Yaskawa INFORM job: OK_R2_O8A-O21A(90,0)OKKR.JBI

/JOB
//NAME OK_R2_O8A-O21A(90,0)OKKR
///FOLDERNAME X4
//POS
///NPOS 663,663,663,26,0,0
///TOOL 0
///POSTYPE PULSE
///PULSE
C00000=132511,-103668,-126871,-1472,79341,68717
C00001=132511,-105453,-125920,-1479,77839,68735
C00002=149942,-121925,-119361,5630,57848,69572
C00003=131289,-120708,-115141,16553,58451,62255
C00004=130492,-107448,-108919,16502,61476,62404
C00005=130492,-107531,-107691,16624,60708,62286
C00006=130492,-107522,-107880,16606,60824,62304
C00007=130122,-101219,-105586,16530,62651,62436
C00008=130467,-107013,-108826,16492,61638,62417
C00009=173804,-84257,-100337,-8034,65857,78258
C00010=173658,-84030,-99866,-7982,65672,78220
C00011=173658,-84451,-98929,-8028,64885,78273
C00012=173658,-84370,-99117,-8019,65041,78263
C00013=172100,-80256,-97322,-7106,65901,77657
C00014=174189,-84275,-102553,-8181,67232,78295
C00015=146680,-106555,-114552,7207,63010,68642
C00016=194694,-79170,-110255,25784,98520,-48468
C00017=198558,-80793,-107909,24687,95396,-47836
C00018=200090,-81195,-106872,24266,94212,-47563
C00019=202263,-84154,-108139,23691,92956,-47080
C00020=202263,-85492,-106716,23644,91519,-47366
C00021=203864,-86202,-108997,23266,92055,-46716
C00022=200090,-81195,-106872,24266,94212,-47563
C00023=174358,-91389,-89628,58384,85447,-80654
C00024=175228,-93280,-90391,58296,84646,-80691
C00025=174358,-91389,-89628,58384,85447,-80654
C00026=168427,-86826,-93699,59246,91643,-79819
C00027=162839,-83719,-106729,43881,81993,-66911
C00028=147123,-91237,-114479,20257,52031,-49855
C00029=112908,-124838,-130477,22240,82773,-36203
C00030=117493,-120147,-121828,21064,78888,-35282
C00031=131517,-88028,-114974,8271,96172,-30135
C00032=131517,-89283,-114090,8245,94996,-30214
C00033=131517,-88930,-114352,8253,95335,-30191
C00034=131178,-82908,-111873,8367,96921,-30191
C00035=131517,-87249,-115462,8285,96867,-30089
C00036=132831,-90163,-114266,11578,93705,-29175
C00037=134095,-89636,-114054,11263,93680,-28777
C00038=131312,-89742,-115220,11972,94693,-29560
C00039=110699,-95947,-121920,22827,92218,-35184
C00040=159423,-136044,-122705,19473,51748,-49954
C00041=156084,-144100,-135379,20578,56007,-50549
C00042=159635,-139405,-132559,18260,112136,-84879
C00043=178843,-153016,-133090,20490,101295,-79475
C00044=178843,-153131,-133279,20494,101347,-79466
C00045=178843,-151887,-131264,20445,100783,-79562
C00046=178843,-153131,-133279,20494,101347,-79466
C00047=178681,-162456,-135669,20227,98263,-80057
C00048=165549,-147119,-131679,18745,106518,-83551
C00049=164263,-165353,-136391,17937,100651,-41944
C00050=168242,-162829,-132237,18538,98565,-40818
C00051=170474,-158220,-131092,19006,99630,-39839
C00052=168242,-162829,-132237,18538,98565,-40818
C00053=163940,-146805,-133599,18623,108164,-40895
C00054=162398,-133850,-130940,19068,113277,-40626
C00055=162571,-113567,-127717,17378,114163,-86924
C00056=160654,-117481,-127396,16916,112431,-87902
C00057=160654,-117651,-127195,16888,112229,-87933
C00058=160654,-118532,-125995,16733,111086,-88103
C00059=160654,-118346,-126273,16766,111343,-88065
C00060=161650,-123459,-127890,16641,109583,-87959
C00061=158594,-113131,-127392,17075,114977,-88272
C00062=174543,-100010,-122844,18621,115499,-82286
C00063=174543,-100010,-122844,18621,115499,-82286
C00064=174543,-100010,-122844,18621,115499,-22315
C00065=138816,-129701,-130055,13678,112254,-36070
C00066=137500,-131474,-125884,13183,109137,-36932
C00067=137500,-131471,-125777,13177,109074,-36939
C00068=139149,-130411,-125460,13458,109147,-36324
C00069=137500,-131471,-125777,13177,109074,-36939
C00070=137500,-129047,-134180,13875,115320,-36192
C00071=137500,-130207,-132407,13667,113680,-36396
C00072=137899,-129904,-132317,13740,113712,-36243
C00073=137899,-129904,-132317,13740,113712,-68510
C00074=153549,-123160,-126704,15778,110958,-63049
C00075=153549,-123239,-126516,15760,110807,-63070
C00076=153549,-123761,-124983,15622,109641,-63231
C00077=153549,-123239,-126516,15760,110807,-63070
C00078=162223,-110280,-122283,17095,113025,-59536
C00079=162223,-111585,-120346,16843,111240,-59807
C00080=163386,-116637,-122034,16744,109515,-59637
C00081=162108,-110157,-121578,17034,112692,-59632
C00082=164629,-100924,-122013,18009,116976,-58006
C00083=164629,-100924,-122013,18009,116976,-86315
C00084=167353,-101147,-115616,17756,113668,-85844
C00085=165427,-104649,-116407,17406,112807,-86697
C00086=165427,-101226,-120322,18070,116786,-86050
C00087=165427,-100996,-120510,18111,117009,-86012
C00088=148525,-143011,-136643,-3983,84771,6637
C00089=128066,-147732,-136598,-30045,86114,11272
C00090=107762,-175532,-134890,-18909,55578,-3499
C00091=107762,-174389,-134000,-18900,55616,-3506
C00092=107762,-171707,-131824,-18892,55653,-3513
C00093=107762,-174389,-134000,-18900,55616,-3506
C00094=110240,-168768,-132692,-19371,58166,-2939
C00095=107762,-174389,-134000,-18900,55616,-3506
C00096=136558,-139033,-124155,-30771,85335,13620
C00097=136645,-139245,-122439,-30816,84359,13917
C00098=135016,-140023,-122655,-30663,83532,13499
C00099=136645,-139245,-122439,-30816,84359,13917
C00100=136645,-142239,-130726,-30739,87441,13088
C00101=136645,-142239,-130726,-30739,87441,13088
C00102=136231,-126717,-125654,-30746,91494,11840
C00103=98133,-136848,-119853,8087,80711,399
C00104=120576,-107226,-130969,-4806,98429,-26759
C00105=134040,-103912,-127141,-12417,95216,-42526
C00106=135128,-102736,-122709,-12628,93295,-41985
C00107=135270,-98410,-119352,-12667,93467,-41957
C00108=135270,-99211,-118697,-12651,92671,-41876
C00109=135270,-98984,-118890,-12655,92901,-41899
C00110=134962,-94751,-117294,-12605,94023,-42111
C00111=135502,-100967,-121058,-12716,93242,-41857
C00112=134459,-102900,-122675,-12466,93098,-42180
C00113=132900,-95838,-124142,-12211,97313,-43092
C00114=133104,-101231,-126476,-12555,90730,-41824
C00115=142488,-103018,-116603,18920,70477,33231
C00116=149408,-93922,-109008,15541,69095,35470
C00117=149408,-94512,-107956,15635,68178,35347
C00118=149408,-94372,-108222,15611,68405,35378
C00119=148690,-90146,-106536,15855,69631,35290
C00120=149408,-93897,-109054,15536,69135,35476
C00121=123067,-90692,-110186,27168,77789,27787
C00122=102416,-91941,-110630,34518,86135,22666
C00123=101917,-92285,-106963,34730,79171,22421
C00124=101917,-92861,-105821,34832,78340,22159
C00125=102166,-91294,-105409,34682,78702,22372
C00126=102552,-87773,-103968,34461,79319,22719
C00127=102166,-90677,-106542,34586,79544,22637
C00128=123117,-127863,-126220,28315,69551,25784
C00129=125315,-122167,-126738,14196,74486,31169
C00130=125647,-109964,-126758,-6698,85320,36650
C00131=127309,-126191,-121158,-24496,77378,41430
C00132=122509,-120998,-116871,-23174,76039,39921
C00133=117160,-104372,-112630,-18566,82677,37125
C00134=117160,-104907,-110988,-18612,81456,37312
C00135=117160,-104733,-111581,-18595,81887,37246
C00136=112842,-111563,-113988,-14481,77147,33000
C00137=113063,-106504,-112219,-14479,78650,32898
C00138=112842,-111563,-113988,-14481,77147,33000
C00139=122612,-110522,-114147,-22924,79491,39282
C00140=127138,-114707,-118233,-24171,81082,40600
C00141=112168,-135147,-125869,-19703,71474,13622
C00142=107112,-124941,-122811,-17686,73526,11445
C00143=98892,-86649,-110918,-2998,94873,-14107
C00144=112057,-63273,-99647,-16927,107898,6848
C00145=111820,-63961,-99109,-16821,107199,6872
C00146=111820,-65039,-98309,-16715,106195,7017
C00147=111820,-64914,-98405,-16727,106313,7000
C00148=110559,-64565,-98232,-16557,106153,6607
C00149=111820,-64402,-98791,-16776,106793,6930
C00150=102401,-90236,-113117,129,94163,-18304
C00151=122722,-94557,-112635,-4536,92169,-11873
C00152=122722,-95060,-112012,-4533,91529,-11850
C00153=122722,-94938,-112169,-4534,91688,-11856
C00154=124421,-94788,-112110,-4914,91823,-11321
C00155=122722,-94458,-112752,-4538,92292,-11877
C00156=121995,-82445,-116286,-4470,100580,-12401
C00157=106227,-105095,-124470,409,77251,-17488
C00158=147196,-120547,-129970,14917,75808,-13222
C00159=161004,-130220,-121828,20444,67155,-12825
C00160=163784,-117907,-115753,19016,68936,-11464
C00161=172766,-99094,-111810,8888,79207,-7928
C00162=172766,-99537,-110960,8908,78464,-7982
C00163=164799,-113448,-113379,18515,69495,-10996
C00164=160173,-111708,-112729,20272,71037,-12446
C00165=159937,-107532,-111273,20230,72269,-12319
C00166=160173,-111708,-112729,20272,71037,-12446
C00167=157530,-113449,-113320,21331,71196,-13397
C00168=157502,-114878,-111335,21583,69377,-13748
C00169=159463,-112600,-110567,20755,69532,-12980
C00170=157502,-114878,-111335,21583,69377,-13748
C00171=157530,-113449,-113320,21331,71196,-13397
C00172=164799,-113448,-113379,18515,69495,-10996
C00173=163784,-117907,-115753,19016,68936,-11464
C00174=161004,-130220,-121828,20444,67155,-12825
C00175=158635,-143974,-124952,47178,64629,48132
C00176=161510,-136095,-119169,46184,63472,49060
C00177=162608,-132555,-115350,46042,62530,49158
C00178=162346,-131008,-113540,46239,62439,48970
C00179=162608,-133192,-116899,45817,62973,49385
C00180=136560,-74570,-80638,73986,100743,31924
C00181=136560,-74368,-74379,73183,99581,30233
C00182=138115,-75223,-74700,73053,98436,30293
C00183=135508,-73752,-74143,73275,100358,30196
C00184=149616,-145660,-96573,81184,49972,24507
C00185=150329,-142641,-96001,80244,49710,25268
C00186=148962,-149729,-97186,82532,50127,23453
C00187=146770,-153464,-99018,82858,51507,22849
C00188=140616,-162996,-103531,83341,55379,21287
C00189=129649,-178931,-115518,81569,62637,20208
C00190=149811,-117254,-127694,14309,93218,9052
C00191=138773,-86779,-112433,16512,101214,6420
C00192=139010,-84837,-109587,16423,100448,6393
C00193=139010,-86284,-108173,16326,98898,6181
C00194=139046,-85929,-108499,16342,99259,6242
C00195=139851,-81484,-106752,16280,100273,6644
C00196=139210,-85073,-109125,16364,100022,6400
C00197=160229,-93267,-112119,12359,94277,12585
C00198=159749,-92653,-111811,12461,94470,12448
C00199=159749,-93339,-110977,12438,93625,12360
C00200=159895,-92298,-111808,12436,94626,12511
C00201=160151,-89339,-110624,12406,95366,12669
C00202=159895,-92298,-111808,12436,94626,12511
C00203=154010,-101242,-121994,13665,97135,10872
C00204=154083,-100267,-121778,13665,97483,10934
C00205=147006,-81102,-116195,13282,100818,-40144
C00206=151269,-63896,-105225,12354,102282,-38687
C00207=152138,-63686,-103764,12097,101397,-38514
C00208=152138,-64898,-103136,12048,100410,-38612
C00209=152138,-64707,-103240,12056,100569,-38597
C00210=153752,-65312,-103536,11647,100239,-38140
C00211=152274,-63472,-103683,12067,101440,-38470
C00212=162010,-107602,-126737,9369,91949,-36281
C00213=162010,-107602,-126737,9369,91949,-36281
C00214=210314,-79584,-107375,-35746,108623,54127
C00215=185587,-33049,-75742,-32288,103518,46434
C00216=184078,-34029,-75535,-31853,102480,46201
C00217=182552,-34930,-76118,-31484,101891,45830
C00218=182816,-34825,-76051,-31547,101988,45895
C00219=182831,-36048,-74896,-31379,100842,46225
C00220=185721,-33305,-75942,-32316,103553,46472
C00221=194611,-82272,-100926,-32769,98332,51304
C00222=192673,-88198,-103442,-32335,96357,51142
C00223=191529,-89685,-104055,-32127,95614,50921
C00224=191825,-89362,-103923,-32180,95794,50983
C00225=191825,-89971,-102555,-32100,94805,51265
C00226=194745,-83421,-100673,-32716,97748,51530
C00227=202657,-68845,-90344,-38048,95727,59775
C00228=197239,-49375,-79846,-37211,96371,57406
C00229=190625,-19292,-60428,-35861,96684,54792
C00230=196048,-18383,-62081,-37469,99924,55713
C00231=194745,-77273,-107470,-33657,103946,49656
C00232=180005,-94840,-122299,4648,94317,-30566
C00233=161456,-138612,-119355,33475,60108,-39853
C00234=177080,-145862,-118570,20687,46862,-30231
C00235=175352,-139433,-111534,22920,46725,-31778
C00236=170439,-155606,-119968,27049,45364,-34664
C00237=142804,-136998,-117626,37100,63175,-22857
C00238=144522,-132180,-113554,36549,62414,-22344
C00239=144766,-128709,-107397,37102,60688,-22883
C00240=136947,-145476,-117578,40176,62334,-25990
C00241=196282,-87995,-108739,3579,85426,-743
C00242=193667,-86961,-103412,6361,79957,-1472
C00243=216929,-66894,-95138,-18936,93102,19193
C00244=189134,-104042,-110891,-11007,79195,11721
C00245=187825,-103632,-110905,-10585,79243,11276
C00246=188383,-103961,-111964,-10748,79789,11413
C00247=188473,-109529,-112575,-10859,77358,11657
C00248=154380,-113917,-114398,722,74096,187
C00249=176928,-85967,-103932,-21600,91605,23275
C00250=179540,-74185,-98826,-24887,98354,27279
C00251=188222,-67873,-108629,-27686,109139,27784
C00252=193624,-62519,-106039,-28903,111697,28985
C00253=181889,-64694,-107206,-10450,102860,-46697
C00254=182813,-61669,-103576,-10649,102295,-46371
C00255=178794,-28814,-84601,-9904,107003,-47957
C00256=175414,-50228,-100699,-8949,105606,-48817
C00257=160705,-81264,-118021,1653,95624,-51077
C00258=127953,-81916,-111881,42691,92562,11616
C00259=120615,-98718,-118071,9470,89242,-10072
C00260=120614,-100809,-115874,9471,86847,-10254
C00261=116758,-96129,-112357,16683,91181,-14824
C00262=119673,-105427,-116369,9746,84913,-10709
C00263=120613,-100772,-115937,9471,86904,-10250
C00264=124245,-107241,-116502,14906,86756,-12895
C00265=120614,-100813,-115850,14161,89229,-15792
C00266=120615,-98722,-118044,14185,91583,-15523
C00267=139593,-120017,-125917,14274,80051,13697
C00268=147459,-122057,-122338,-8250,71740,26203
C00269=147460,-122349,-119714,-8332,69994,26324
C00270=147216,-123530,-118779,-8298,68797,26321
C00271=147775,-127178,-120450,-8566,68018,26578
C00272=149021,-123014,-119622,-8969,69764,26896
C00273=148272,-123606,-115899,-8821,67114,26825
C00274=147464,-122345,-117274,-8412,68510,26430
C00275=147464,-122366,-119995,-8326,70156,26314
C00276=147464,-118224,-129513,-8030,78063,25782
C00277=147464,-118224,-129513,-6689,118601,78925
C00278=147464,-118224,-129513,-6689,118601,90375
C00279=129716,-111878,-123336,3524,122371,86039
C00280=131368,-111986,-122768,3938,121897,86671
C00281=90490,-99752,-122446,-25205,102120,77013
C00282=92153,-96107,-120269,-25526,103067,77386
C00283=127155,-108660,-119184,2836,121576,85017
C00284=126355,-98414,-119449,2829,127024,84850
C00285=140836,-122858,-129041,139,116760,83504
C00286=140645,-125315,-128438,105,115126,83435
C00287=121833,-132425,-113961,-44925,89262,78761
C00288=121169,-125555,-111250,-44945,90266,78000
C00289=151886,-132757,-130646,2140,112507,87535
C00290=173213,-138110,-133115,-4817,110614,73303
C00291=178695,-122684,-126329,-7235,117632,76997
C00292=178664,-97821,-112009,32036,94837,77481
C00293=178457,-102445,-114055,32005,93957,77153
C00294=183114,-120871,-123216,-6165,117012,78717
C00295=183838,-120175,-121246,-5947,116214,79037
C00296=182806,-113441,-126130,-6638,122566,78264
C00297=165277,-120173,-132750,-1498,117651,75946
C00298=166684,-149732,-138114,9906,98033,76858
C00299=201464,-114352,-117147,5757,101650,-67438
C00300=200368,-109540,-114804,5783,102752,-67759
C00301=168812,-128354,-130665,8728,111437,78365
C00302=168516,-129586,-131473,-968,112075,77186
C00303=152590,-129390,-129911,-3156,110818,71484
C00304=141826,-124162,-127188,-4588,111325,67607
C00305=141114,-115628,-126239,-4831,115072,67194
C00306=147247,-120038,-130806,8856,110749,89640
C00307=138147,-116215,-122144,16955,111448,87520
C00308=136269,-107535,-118257,19196,116051,87125
C00309=188488,-115235,-117264,-8764,104512,-67856
C00310=187301,-109373,-114560,-8881,105718,-68358
C00311=135583,-106226,-116474,19024,115804,86815
C00312=137886,-102725,-119104,19994,118513,88211
C00313=139135,-112852,-128624,20291,118843,88765
C00314=139292,-114870,-129287,20177,118215,88704
C00315=187982,-104318,-127456,-3477,89797,-72703
C00316=187990,-108723,-124740,-3481,85869,-72593
C00317=186449,-106135,-122224,-3009,85591,-73073
C00318=188099,-109945,-124726,-3517,85239,-72540
C00319=187395,-105029,-122279,-3298,86229,-72790
C00320=187063,-105219,-121972,-3196,85930,-72888
C00321=188029,-108820,-124772,-3493,85841,-72579
C00322=188022,-104421,-127490,-3489,89767,-72690
C00323=174298,-113219,-115861,15770,66124,24057
C00324=181162,-106311,-114496,5429,75659,20720
C00325=173939,-113739,-113379,16158,64464,23688
C00326=174688,-117897,-113404,16083,62276,23658
C00327=177951,-106650,-114504,8052,76050,18386
C00328=176740,-112744,-108858,15100,61741,24377
C00329=174039,-113317,-109052,16445,62092,23376
C00330=173285,-113495,-108535,16870,61851,23047
C00331=174267,-113511,-110133,16253,62591,23541
C00332=174258,-113480,-112891,16028,64241,23777
C00333=174307,-102252,-117157,11533,81046,15470
C00334=174345,-102365,-117198,11521,81009,15479
C00335=190775,-91857,-121708,-11796,95177,30723
C00336=208754,-98864,-112717,-37128,92966,49075
C00337=214846,-120327,-106837,-51151,83157,62011
C00338=214841,-119670,-104864,-51217,82591,62323
C00339=213604,-125439,-105942,-50991,78248,62021
C00340=216770,-120620,-104459,-51433,83201,63007
C00341=216373,-116987,-103296,-51322,83714,62508
C00342=214193,-116769,-100356,-51274,81398,62635
C00343=214845,-118750,-102310,-51312,81889,62717
C00344=214851,-119483,-104312,-51238,82440,62412
C00345=218178,-115538,-118233,-49266,91982,56948
C00346=169784,-95533,-109053,-46596,84452,-16696
C00347=175845,-105369,-102937,-51834,73714,-22623
C00348=175640,-91669,-95359,-54212,78616,-24875
C00349=173505,-93584,-96126,-53785,77091,-25122
C00350=169740,-90290,-95011,-54323,79351,-24910
C00351=170527,-92138,-98060,-54392,80356,-25101
C00352=164897,-89030,-99124,-48240,79718,-32152
C00353=161372,-116003,-107175,-47183,64470,-24730
C00354=161496,-116499,-106623,-47427,64124,-24479
C00355=159887,-93001,-100921,-46911,76509,-32980
C00356=98520,-84299,-97494,-15890,55411,-52136
C00357=162881,-120047,-112782,-46142,67476,-23200
C00358=153966,-116641,-122556,-34655,76025,-15464
C00359=117008,-148876,-136987,1466,73673,38063
C00360=126252,-131765,-130839,-5463,89111,40743
C00361=118320,-126497,-124056,-4164,87185,38181
C00362=118819,-79314,-106757,-4355,100773,37882
C00363=119819,-85991,-113186,-4537,101348,38176
C00364=122079,-96641,-122243,-4925,101568,38878
C00365=101099,-87648,-113482,27968,109543,-44429
C00366=120135,-78703,-106739,14797,112831,-39871
C00367=120170,-67936,-101208,14266,107328,-40543
C00368=110218,-114507,-123212,16108,86718,-46162
C00369=152504,-138441,-132085,-16664,78093,9085
C00370=191457,-109567,-125034,-9426,80684,19151
C00371=214381,-113602,-114057,-27955,63726,64142
C00372=214387,-113723,-111179,-28386,62102,64581
C00373=215427,-113571,-109853,-29050,61806,65105
C00374=214389,-113728,-111258,-28375,62143,64570
C00375=212738,-111566,-109277,-27620,61502,64048
C00376=215080,-114206,-110031,-28945,61493,65044
C00377=214706,-116049,-110700,-28908,60895,65052
C00378=214364,-113704,-111171,-28374,62098,64572
C00379=214357,-113582,-114048,-27943,63722,64133
C00380=174283,-101247,-119871,-16121,93821,65453
C00381=174399,-103758,-119266,-16107,92243,65697
C00382=173872,-98338,-116871,-16021,93408,65372
C00383=175145,-99456,-118673,-16315,94157,65691
C00384=175025,-104520,-116447,-20806,93585,64920
C00385=174312,-103656,-117420,-20719,94391,64539
C00386=176714,-116929,-126906,-19302,86766,16179
C00387=181382,-121683,-127165,5388,71552,36447
C00388=187446,-131805,-111566,37879,40004,62235
C00389=187463,-129896,-107666,38934,38872,61621
C00390=198864,-139275,-106761,28144,24177,62608
C00391=186446,-131716,-107742,40356,38644,60793
C00392=185573,-127298,-105247,40377,39617,60774
C00393=197435,-137317,-104978,29287,25809,64127
C00394=187457,-128566,-105102,39647,38173,61211
C00395=187441,-130558,-109037,38564,39279,61835
C00396=196640,-143323,-122728,29866,37120,66734
C00397=185945,-125174,-129582,39897,103153,69319
C00398=193646,-124792,-118080,38663,94346,69340
C00399=212686,-113481,-89566,12963,78888,-71132
C00400=215151,-115296,-90915,12760,78396,-70316
C00401=198243,-108662,-112800,38731,96308,72004
C00402=197696,-107272,-114471,38964,97919,72363
C00403=152343,-113083,-118185,24814,126675,56048
C00404=153493,-118526,-118240,24301,123820,55827
C00405=215589,-109296,-82766,10801,104809,-70870
C00406=212839,-110161,-82796,9951,104741,-71860
C00407=156810,-114950,-114235,25206,122271,56916
C00408=155394,-107237,-115802,26414,127157,57611
C00409=147814,-144132,-130264,24847,111600,50742
C00410=214385,-115050,-91121,15616,71856,-39505
C00411=214401,-113114,-87216,15735,70495,-39681
C00412=214407,-112311,-85637,15785,69955,-39751
C00413=212607,-111613,-85852,16057,70779,-40304
C00414=214366,-115000,-87352,15823,69648,-39808
C00415=214392,-111585,-84244,16055,65381,-44584
C00416=214410,-109897,-81022,24415,69187,-61260
C00417=214414,-110066,-81336,23540,70296,-59097
C00418=214409,-110914,-82947,23467,70808,-58993
C00419=214399,-112969,-86931,23295,72098,-58733
C00420=182860,-108511,-132060,8820,106503,33858
C00421=240778,-137351,-128254,-45983,85020,-28938
C00422=236675,-121649,-106302,-61967,62621,-57515
C00423=232044,-114198,-104885,-58168,72082,-54237
C00424=230371,-110875,-95735,-61232,57885,-58042
C00425=229315,-118320,-101960,-58791,68287,-53156
C00426=229655,-120240,-104287,-58708,68736,-53276
C00427=234952,-97476,-90701,-63445,70634,-56635
C00428=230316,-114034,-100213,-59700,68809,-54050
C00429=229268,-118961,-102390,-58804,68223,-53138
C00430=229453,-118187,-100297,-59129,67859,-52730
C00431=229511,-117701,-99692,-59180,67829,-52669
C00432=228007,-118154,-101138,-58697,67254,-53236
C00433=227998,-119492,-104806,-58168,68101,-53893
C00434=217117,-124631,-136943,-31097,89965,-17175
C00435=212311,-124866,-133165,-25299,83870,-9309
C00436=196995,-84615,-117906,17381,99261,54937
C00437=196689,-87191,-114654,17284,96138,54393
C00438=196190,-85752,-112362,17378,95592,54154
C00439=196743,-87074,-114185,17262,95909,54377
C00440=198014,-90395,-114090,16887,93977,54517
C00441=205154,-51487,-95949,15259,101027,57955
C00442=205373,-53531,-98850,15247,101700,58106
C00443=205704,-49963,-101444,15409,104963,58624
C00444=178318,-108601,-128727,5603,100252,45769
C00445=168853,-122238,-134242,1220,95726,41713
C00446=170297,-107383,-120290,-24028,103073,37740
C00447=160733,-103929,-113030,-25314,98004,34995
C00448=161047,-105663,-112613,-25510,98022,34157
C00449=162344,-106453,-112811,-25592,98148,34602
C00450=160733,-103887,-113137,-25583,99045,33815
C00451=160980,-105138,-113190,-19033,89916,22163
C00452=160982,-105109,-112996,-20911,91648,19194
C00453=152566,-110009,-113460,3309,75991,4288
C00454=157788,-107819,-112956,241,74994,7914
C00455=120609,-111596,-118782,-13024,86064,14317
C00456=133998,-113178,-111834,-29794,79414,36692
C00457=133784,-113259,-111042,-29784,78878,36749
C00458=133610,-109140,-109688,-29638,79939,36406
C00459=135828,-112441,-110974,-30250,79928,37264
C00460=134042,-113729,-112572,-24695,80409,36334
C00461=133994,-113037,-113381,-24636,81174,36157
C00462=133996,-112670,-115866,-24554,82743,35831
C00463=134898,-132336,-126413,-10595,74184,11936
C00464=133962,-121152,-121142,2699,71953,-10515
C00465=133963,-121408,-118595,2724,70256,-10553
C00466=134171,-122182,-117969,2655,69467,-10496
C00467=132452,-124377,-118846,3342,68943,-11121
C00468=134389,-126169,-119210,2591,68176,-10448
C00469=130565,-111827,-114257,5039,75994,-15555
C00470=126623,-133823,-126710,6462,72649,-17071
C00471=133973,-119339,-126131,2645,75950,-10424
C00472=158112,-98716,-126250,19680,86530,48527
C00473=161036,-120263,-128161,18992,76528,47904
C00474=161025,-122948,-118687,19668,69709,46778
C00475=160677,-121425,-116341,19892,69174,46554
C00476=161739,-127404,-118540,19698,67291,46630
C00477=160544,-119732,-117016,19776,70412,46719
C00478=170277,-111094,-113056,15772,70241,50261
C00479=171080,-122297,-124815,15314,71519,50716
C00480=162896,-130847,-128779,13430,60460,45398
C00481=130949,-94872,-120528,-14594,85248,55395
C00482=53825,-116322,-125048,14351,65953,45020
C00483=-30260,-81955,-85592,10541,58194,-89907
C00484=126253,-78535,-68629,1974,68777,-60728
C00485=133976,-48579,-51749,422,66953,-55442
C00486=143445,-11852,-31053,-1480,64717,-48962
C00487=147670,17027,-9476,-9877,74622,-49123
C00488=147135,31900,7029,-9795,72081,-49101
C00489=147059,31291,7516,-9797,71470,-49078
C00490=147059,31341,6529,-9765,72092,-49129
C00491=147727,26207,1471,-9995,72641,-48940
C00492=147727,26139,2513,-10029,71973,-48885
C00493=147511,27771,4102,-9954,71808,-48945
C00494=147650,25585,2035,-9999,71973,-48912
C00495=147650,26097,-2600,-9851,75043,-49164
C00496=119782,42933,14409,-5087,72220,-53475
C00497=118099,48860,22276,-4468,70330,-53985
C00498=118099,48825,24454,-4506,68976,-53934
C00499=118090,47987,23851,-4504,68915,-53935
C00500=118090,48004,24664,-4522,68425,-53913
C00501=118090,47958,23810,-4504,68925,-53935
C00502=118049,44181,19766,-4472,69469,-53971
C00503=118049,44151,20600,-4487,68943,-53949
C00504=118075,46427,23028,-4508,68620,-53926
C00505=118049,44122,20560,-4487,68953,-53949
C00506=118049,44425,14984,-4396,72529,-54081
C00507=116860,-24994,-46486,-3887,74622,-54555
C00508=141580,-19095,-42244,-13161,77572,-46437
C00509=154421,-19095,-42244,7152,69599,-54311
C00510=168772,13045,-11724,355,66689,-49386
C00511=168772,13045,-11724,355,66689,-49386
C00512=178887,35491,12589,-4659,63528,-45673
C00513=181596,22371,-6368,6207,82852,-43396
C00514=181122,23764,-2510,5908,81004,-43496
C00515=181122,23670,-1654,5914,80431,-43522
C00516=181122,23764,-2510,5908,81004,-43496
C00517=178663,19949,-6903,6582,81925,-44269
C00518=179355,21466,-3674,6406,80670,-44103
C00519=179829,21504,-3239,6279,80388,-43959
C00520=178670,19793,-5916,6590,81240,-44302
C00521=173498,18801,-6845,8008,81758,-45996
C00522=173844,18831,-3651,7950,79792,-46005
C00523=173838,18807,-2614,7966,79149,-46049
C00524=173844,18768,-1984,7975,78746,-46073
C00525=173844,18778,-2337,7967,78964,-46058
C00526=174883,21039,-87,7686,78645,-45722
C00527=173850,18758,-2365,7965,78970,-46055
C00528=173850,19604,-9778,7879,83922,-45740
C00529=173850,19604,-9778,7879,54886,-45740
C00530=178844,-3710,-18963,4726,48213,-44074
C00531=169145,-109680,-85477,15638,36065,-50412
C00532=234460,-155557,-97015,-52723,35880,-9269
C00533=234460,-155557,-97015,-52723,35880,-9269
C00534=233592,-182620,-119845,-52271,35507,-9647
C00535=185005,-180970,-119127,-52124,36225,-9601
C00536=146370,-47178,-55409,-22603,47358,-44094
C00537=150355,38217,32552,-52662,46329,-47179
C00538=136449,20180,17702,-29375,35603,-50157
C00539=135403,43871,52603,-36669,27312,-46380
C00540=135403,44850,54869,-37729,26595,-45848
C00541=135403,44693,54509,-37558,26707,-45934
C00542=135667,46652,56638,-38197,26579,-45595
C00543=135403,43905,52678,-36703,27288,-46362
C00544=136689,45067,54900,-38900,27228,-45168
C00545=138426,130785,55808,-24075,105508,-62741
C00546=138672,133033,60852,-23888,103779,-62297
C00547=136689,45067,54900,-38900,27228,-45168
C00548=133482,49096,59308,-36365,25336,-46668
C00549=134347,38712,45394,-33634,28355,-47978
C00550=116454,-24761,-39686,-5990,62430,-55725
C00551=125251,-119211,-114122,-8766,63875,-48424
C00552=166025,-25947,-80013,-26532,97101,-31760
C00553=164294,-17063,-34958,31065,55273,54461
C00554=168124,42014,10128,23159,81576,60225
C00555=168124,42014,10128,23159,81576,60225
C00556=172413,73393,40128,13737,95185,62195
C00557=173406,55787,34570,11199,81413,60765
C00558=173520,53424,33189,11186,81039,60771
C00559=172413,73393,40128,13737,95185,62195
C00560=174432,74681,41670,13553,94577,62815
C00561=169243,43363,4993,17420,85083,59919
C00562=175926,65443,14304,7549,79996,66162
C00563=173251,57933,12957,12377,73806,65557
C00564=175037,96499,49818,7828,90248,66438
C00565=175152,93287,46964,7802,90342,66481
C00566=173251,57933,12957,12377,73806,65557
C00567=175259,59080,14259,11439,73326,66178
C00568=173823,64435,15621,8474,78871,65427
C00569=163328,22111,-17695,16319,60605,55206
C00570=158063,-10254,-35326,-2776,53207,35705
C00571=177458,-62225,-50397,-53512,41611,19716
C00572=174476,-83233,-86994,-43003,48026,24087
C00573=139045,-11347,-51706,-12836,64434,-19988
C00574=127239,32842,15043,-2972,60837,-63802
C00575=119734,32558,24909,4032,51838,-73141
C00576=129950,39474,50975,-5681,27732,-67581
C00577=135865,87011,40718,-24918,95497,-56957
C00578=136153,89985,46203,-24876,93896,-56517
C00579=129761,47736,62677,-6046,24776,-67415
C00580=132478,43229,57759,-9474,25736,-65476
C00581=129950,39474,50975,-5681,27732,-67581
C00582=131685,-19323,-9200,-7335,35490,-65222
C00583=102327,-132081,-105905,9820,46482,-54731
C00584=168046,-22646,-92303,-23676,100531,-31319
C00585=178506,-64043,-51330,-54345,42002,9320
C00586=161820,24023,-17780,7570,61243,60628
C00587=163544,81139,32356,1868,89449,65267
C00588=166900,113245,76474,-383,92426,67637
C00589=158379,103529,59182,8519,87603,65182
C00590=158357,100044,55900,8524,87832,65191
C00591=165104,112461,75430,-214,92658,67037
C00592=163544,81139,32356,1868,89449,65267
C00593=164280,62524,18315,-3678,70871,65511
C00594=166828,64073,25097,-5062,67634,66495
C00595=143537,101175,57606,16851,87230,68252
C00596=143394,97839,54544,16884,87421,68231
C00597=164844,63557,24497,-4043,67628,65806
C00598=164280,62524,18315,-3678,70871,65511
C00599=158520,39777,460,10756,55186,64462
C00600=156529,-359,-32075,-2996,54939,55409
C00601=181545,-68424,-52291,-57183,42847,45278
C00602=151832,-108617,-86131,-35646,27145,3822
C00603=153330,-47816,-46612,-35487,59555,-26701
C00604=157028,39295,61974,-48386,44011,-18265
C00605=155433,37642,66776,-34947,32543,-17522
C00606=140151,91077,43318,5378,90823,-76333
C00607=140389,94148,48975,5317,88913,-76337
C00608=159561,37168,66275,-37223,34214,-15663
C00609=156514,28846,54897,-33266,35284,-18273
C00610=151117,-9182,12555,-27217,39927,-22318
C00611=173224,18806,36696,-37861,47924,-13334
C00612=169464,28118,25687,-11023,65897,-4984
C00613=169711,38038,41079,-11502,61638,-4466
C00614=169887,43923,50617,-11874,58875,-4105
C00615=186672,90586,45814,14233,85155,71230
C00616=186465,93628,48420,14293,85151,71161
C00617=166601,42750,49362,-10823,58586,-5370
C00618=167386,32759,35664,-10728,61929,-5392
C00619=171949,41386,44413,5394,60596,-4250
C00620=171325,51919,57132,7927,61010,-4612
C00621=171177,53470,59840,8034,60163,-4729
C00622=173162,91192,47015,26597,96822,52438
C00623=173064,94370,49802,26605,96778,52392
C00624=174688,55674,62330,7067,59444,-3425
C00625=169529,36419,34103,8013,67341,-4841
C00626=169529,36419,34103,8013,67341,88465
C00627=169151,51771,52338,12064,69022,88341
C00628=169444,62384,65518,10661,69426,88585
C00629=162801,94753,47772,7506,90872,66819
C00630=162783,98187,53928,7502,88866,66693
C00631=173780,65299,68932,10048,68280,90052
C00632=169735,59480,57290,10411,72898,88997
C00633=183539,66276,65186,8173,69882,83660
C00634=183524,67999,71925,8353,66654,83428
C00635=185377,71138,75692,8069,65768,84041
C00636=183464,63606,61545,8145,70748,83691
C00637=183464,63606,61545,8145,70748,10436
C00638=183427,70838,75684,8423,65818,10075
C00639=183567,76740,84490,8560,63442,9952
C00640=161324,95565,53507,9580,75474,63025
C00641=161323,99500,60299,9673,73346,62856
C00642=185394,80422,89094,8298,62324,10546
C00643=183022,56506,58410,8307,69091,10164
C00644=165276,5967,-41282,8150,81970,62723
C00645=150783,-9649,-54161,14441,83650,58478
C00646=92014,-65792,-98652,33579,68908,44779
C00647=112544,25072,-21983,21189,62436,50668
C00648=133924,64642,16887,41400,76255,73236
C00649=139901,71761,28474,30769,75742,73566
C00650=139687,75607,37002,31287,72996,72717
C00651=141837,73425,34521,30373,72588,73444
C00652=143156,96915,63460,30855,67143,72441
C00653=145100,103355,67895,23032,69595,73065
C00654=145405,107585,71935,19869,70388,73011
C00655=142867,98447,59319,20505,73887,72688
C00656=136885,86681,52237,36281,86528,76665
C00657=135724,73725,40183,40167,80560,75024
C00658=136738,86799,56264,40254,77639,74339
C00659=134674,77415,38418,40217,83337,75634
C00660=126958,42470,-7112,42423,94399,76801
C00661=124399,-38669,-81065,43564,98333,77427
C00662=15465,-107351,-121619,48207,78518,35388
BC00000=166335,472416,1075065
BC00001=124697,353752,1075065
BC00002=68977,283557,1075139
BC00003=68977,283557,1075139
BC00004=68977,283557,1075139
BC00005=68977,283557,1075139
BC00006=68977,283557,1075139
BC00007=68977,283557,1075139
BC00008=68977,283557,1075139
BC00009=68977,283557,1075139
BC00010=68978,283557,1075135
BC00011=68978,283557,1075135
BC00012=68978,283557,1075135
BC00013=68978,283557,1075135
BC00014=68978,283557,1075135
BC00015=68977,283557,1075139
BC00016=168951,309918,1075139
BC00017=168951,309918,1075139
BC00018=168951,309918,1075139
BC00019=168951,309918,1075139
BC00020=168951,309918,1075139
BC00021=168951,309918,1075139
BC00022=168951,309918,1075139
BC00023=168951,309918,1075139
BC00024=168951,309918,1075139
BC00025=168951,309918,1075139
BC00026=168951,309918,1075139
BC00027=173594,303876,1075139
BC00028=182502,292282,1075139
BC00029=137284,247060,1075139
BC00030=137284,247060,1075139
BC00031=137284,247060,1075139
BC00032=137284,247060,1075139
BC00033=137284,247060,1075139
BC00034=137284,247060,1075139
BC00035=137284,247060,1075139
BC00036=137284,247060,1075139
BC00037=137284,247060,1075139
BC00038=137284,247060,1075139
BC00039=137284,247060,1075139
BC00040=206498,230878,1075139
BC00041=206498,230878,1075139
BC00042=192552,150198,1075139
BC00043=190994,154806,1075139
BC00044=190994,154806,1075139
BC00045=190994,154806,1075139
BC00046=190994,154806,1075139
BC00047=190994,154806,1075139
BC00048=190994,154806,1075139
BC00049=199392,154806,1075139
BC00050=199392,154806,1075139
BC00051=199392,154806,1075139
BC00052=199392,154806,1075139
BC00053=199392,154806,1075139
BC00054=249664,154806,1075136
BC00055=249665,154806,1075133
BC00056=249665,154806,1075133
BC00057=249665,154806,1075133
BC00058=249665,154806,1075133
BC00059=249665,154806,1075133
BC00060=249665,154806,1075133
BC00061=249665,154806,1075133
BC00062=249665,154806,1075133
BC00063=249665,154806,1075133
BC00064=249665,154806,1075133
BC00065=249665,154806,1075133
BC00066=249665,154806,1075133
BC00067=249665,154806,1075133
BC00068=249665,154806,1075133
BC00069=249665,154806,1075133
BC00070=249665,154806,1075182
BC00071=249437,328326,1075133
BC00072=249437,328326,1075133
BC00073=249437,328326,1075133
BC00074=249437,328326,1075133
BC00075=249437,328326,1075133
BC00076=249437,328326,1075133
BC00077=249437,328326,1075133
BC00078=249437,328326,1075133
BC00079=249437,328326,1075133
BC00080=249437,328326,1075133
BC00081=249437,328326,1075133
BC00082=249437,328326,1075133
BC00083=249437,328326,1075133
BC00084=249437,328326,1075130
BC00085=249437,328326,1075130
BC00086=249437,328326,1075130
BC00087=249437,328326,1075162
BC00088=167636,332713,1075160
BC00089=42922,318475,1073860
BC00090=42922,318475,1073860
BC00091=42922,318475,1073860
BC00092=42922,318475,1073860
BC00093=42922,318475,1073860
BC00094=42922,318475,1073860
BC00095=42922,318475,1073860
BC00096=42922,318475,1073860
BC00097=42922,318475,1073860
BC00098=42922,318475,1073860
BC00099=42922,318475,1073860
BC00100=42922,318475,1073860
BC00101=211008,318519,1073860
BC00102=211008,318519,1073860
BC00103=216837,311609,1073968
BC00104=207508,258847,1074700
BC00105=201911,227194,1075139
BC00106=201911,227194,1075139
BC00107=201911,227194,1075139
BC00108=201911,227194,1075139
BC00109=201911,227194,1075139
BC00110=201911,227194,1075139
BC00111=201911,227194,1075139
BC00112=201911,227194,1075139
BC00113=201911,227194,1075139
BC00114=203477,244762,1075139
BC00115=350651,232694,1075139
BC00116=350651,232694,1075137
BC00117=350651,232694,1075137
BC00118=350651,232694,1075137
BC00119=350651,232694,1075137
BC00120=350651,232694,1075137
BC00121=350651,232694,1075139
BC00122=350651,232694,1075139
BC00123=350651,232694,1075139
BC00124=350651,232694,1075139
BC00125=350651,232694,1075139
BC00126=350651,232694,1075139
BC00127=350651,232694,1075139
BC00128=350651,232694,1075139
BC00129=334060,231848,1075139
BC00130=306342,230434,1075139
BC00131=283190,229253,1075139
BC00132=283190,229253,1075139
BC00133=283190,229253,1075139
BC00134=283190,229253,1075139
BC00135=283190,229253,1075139
BC00136=283190,229253,1075139
BC00137=283190,229253,1075139
BC00138=283190,229253,1075139
BC00139=283190,229253,1075139
BC00140=283190,229253,1075139
BC00141=292053,239754,1075139
BC00142=292053,239754,1075139
BC00143=338604,314190,1075139
BC00144=338604,314190,1075139
BC00145=338604,314190,1075139
BC00146=338604,314190,1075139
BC00147=338604,314190,1075139
BC00148=338604,314190,1075139
BC00149=338604,314190,1075139
BC00150=338604,314190,1075139
BC00151=338604,314190,1075139
BC00152=338604,314190,1075139
BC00153=338604,314190,1075139
BC00154=338604,314190,1075139
BC00155=338604,314190,1075139
BC00156=338604,314190,1075139
BC00157=304912,249417,1075139
BC00158=308898,253323,1075138
BC00159=310242,254639,1075139
BC00160=310242,254639,1075139
BC00161=310242,254639,1075139
BC00162=310242,254639,1075139
BC00163=310242,254639,1075139
BC00164=310242,254639,1075139
BC00165=310242,254639,1075139
BC00166=310242,254639,1075139
BC00167=310242,254639,1075139
BC00168=310242,254639,1075139
BC00169=310242,254639,1075139
BC00170=310242,254639,1075139
BC00171=310242,254639,1075139
BC00172=310242,254639,1075139
BC00173=310242,254639,1075139
BC00174=310242,254639,1075139
BC00175=123796,340399,1075139
BC00176=123796,340399,1075139
BC00177=123796,340399,1075139
BC00178=123796,340399,1075139
BC00179=123796,340399,1075139
BC00180=123796,340399,1075139
BC00181=123796,340399,1075139
BC00182=123796,340399,1075139
BC00183=123796,340399,1075139
BC00184=123796,340399,1075139
BC00185=123796,340399,1075139
BC00186=123796,340399,1075139
BC00187=123796,340399,1075139
BC00188=123796,340399,1075139
BC00189=123796,340399,1075139
BC00190=123796,340399,1075139
BC00191=123796,340399,1075139
BC00192=123796,340399,1075139
BC00193=123796,340399,1075139
BC00194=123796,340399,1075139
BC00195=123796,340399,1075139
BC00196=123796,340399,1075139
BC00197=123796,340399,1075139
BC00198=123796,340399,1075139
BC00199=123796,340399,1075139
BC00200=123796,340399,1075139
BC00201=123796,340399,1075139
BC00202=123796,340399,1075139
BC00203=123796,340399,1075139
BC00204=123796,340399,1075139
BC00205=123796,340399,1075139
BC00206=123796,340399,1075139
BC00207=123796,340399,1075139
BC00208=123796,340399,1075139
BC00209=123796,340399,1075139
BC00210=123796,340399,1075139
BC00211=123796,340399,1075139
BC00212=123796,340399,1075139
BC00213=39157,402685,1075139
BC00214=39157,402685,1075139
BC00215=39157,402685,1075139
BC00216=39157,402685,1075139
BC00217=39157,402685,1075139
BC00218=39157,402685,1075139
BC00219=39157,402685,1075139
BC00220=39157,402685,1075139
BC00221=39157,402685,1075139
BC00222=39157,402685,1075139
BC00223=39157,402685,1075139
BC00224=39157,402685,1075139
BC00225=39157,402685,1075139
BC00226=39157,402685,1075139
BC00227=66315,407376,1075139
BC00228=66315,407376,1075139
BC00229=66315,407376,1075139
BC00230=66315,407376,1075139
BC00231=39157,402685,1075139
BC00232=123796,340399,1075139
BC00233=123796,340399,1075139
BC00234=123796,340399,1075139
BC00235=123796,340399,1075135
BC00236=123796,340399,1075135
BC00237=141932,338819,1075136
BC00238=141932,338819,1075136
BC00239=141932,338819,1075136
BC00240=141932,338819,1075136
BC00241=141932,338819,1075136
BC00242=141932,338819,1075136
BC00243=141932,338819,1075136
BC00244=141932,338819,1075136
BC00245=141932,338819,1075136
BC00246=141932,338819,1075136
BC00247=141932,338819,1075136
BC00248=141932,338819,1075136
BC00249=141932,338819,1075136
BC00250=141932,338819,1075136
BC00251=141932,338819,1075136
BC00252=141932,338819,1075136
BC00253=141932,338819,1075136
BC00254=141932,338819,1075136
BC00255=141932,338819,1075136
BC00256=141932,338819,1075136
BC00257=141932,338819,1075136
BC00258=176377,335818,1075139
BC00259=222039,289329,1075139
BC00260=219738,284348,1075139
BC00261=226738,277671,1075138
BC00262=218817,282356,1075139
BC00263=218817,282356,1075139
BC00264=226738,277671,1075139
BC00265=221524,283439,1075139
BC00266=224948,287784,1075139
BC00267=248818,285296,1075139
BC00268=216295,295930,1075139
BC00269=217822,290313,1075139
BC00270=218433,288066,1075139
BC00271=218433,288066,1075139
BC00272=218433,288066,1075139
BC00273=215305,289815,1075139
BC00274=214546,292145,1075139
BC00275=213019,297762,1075139
BC00276=213019,297762,1075139
BC00277=213019,297762,1075139
BC00278=213019,159800,1075139
BC00279=213019,159800,1075139
BC00280=213019,159802,1075139
BC00281=114731,245528,1036586
BC00282=114731,245528,1036586
BC00283=213019,159800,1075139
BC00284=213019,159800,1075139
BC00285=213019,159800,1075139
BC00286=213019,159800,1075139
BC00287=108147,249003,1075139
BC00288=108147,249003,1075139
BC00289=213019,159800,1075139
BC00290=213019,159800,1075139
BC00291=213019,159800,1075139
BC00292=317009,206720,1075139
BC00293=317009,206720,1075139
BC00294=213019,159800,1075139
BC00295=213019,159800,1075139
BC00296=213019,159800,1075139
BC00297=139063,207884,1075139
BC00298=139064,217157,1072913
BC00299=214976,229852,1075139
BC00300=214976,229852,1075139
BC00301=139063,207884,1072911
BC00302=139063,207884,1072911
BC00303=139063,207884,1072911
BC00304=139063,207884,1072911
BC00305=139063,207884,1072911
BC00306=179195,200940,1072911
BC00307=179195,200940,1074134
BC00308=179195,200940,1074134
BC00309=161162,274129,1075139
BC00310=161162,274129,1075139
BC00311=179195,200940,1074134
BC00312=179195,200940,1074134
BC00313=179195,194430,1074134
BC00314=246753,324307,1074134
BC00315=94933,340328,1075139
BC00316=94225,340492,1075139
BC00317=93948,340556,1075139
BC00318=93942,340557,1075139
BC00319=93942,340557,1075139
BC00320=74466,351481,1075139
BC00321=74750,351415,1075139
BC00322=75457,351251,1075139
BC00323=233051,306144,1075139
BC00324=197054,309147,1075139
BC00325=228471,299468,1075139
BC00326=228471,299468,1075139
BC00327=220252,296135,1075139
BC00328=254158,285052,1075139
BC00329=254158,285052,1075137
BC00330=254158,285052,1075137
BC00331=255466,286960,1075139
BC00332=258738,291728,1075139
BC00333=225045,302219,1075139
BC00334=201847,315231,1075139
BC00335=178964,320129,1075139
BC00336=153924,325488,1075139
BC00337=139402,328596,1075139
BC00338=142990,322553,1075139
BC00339=144424,320136,1075139
BC00340=144424,320136,1075139
BC00341=144424,320136,1075139
BC00342=144422,320132,1075139
BC00343=142987,322549,1075139
BC00344=139400,328591,1075139
BC00345=144112,325650,1075139
BC00346=253442,257415,1075139
BC00347=273235,245062,1075139
BC00348=273235,245062,1075139
BC00349=273235,245062,1075139
BC00350=273235,245062,1075139
BC00351=273235,245062,1075139
BC00352=273637,242934,1075139
BC00353=273901,241536,1075139
BC00354=273901,241536,1075139
BC00355=273637,242934,1075139
BC00356=273637,242934,1075139
BC00357=365806,226163,1075139
BC00358=376725,229265,1075139
BC00359=370640,245115,1075139
BC00360=370640,298070,1075139
BC00361=370640,298070,1075139
BC00362=370640,298070,1075139
BC00363=370640,298070,1075139
BC00364=370640,298070,1075139
BC00365=370640,298070,1075139
BC00366=370640,298070,1075139
BC00367=370640,298070,1075139
BC00368=370640,298070,1075139
BC00369=386406,271889,1075139
BC00370=361249,231483,1075139
BC00371=315377,202556,1075139
BC00372=315063,197107,1075139
BC00373=314939,194954,1075139
BC00374=314938,194928,1075139
BC00375=314938,194928,1075139
BC00376=319640,194110,1075139
BC00377=323135,193503,1075139
BC00378=324656,195440,1075139
BC00379=324969,200889,1075139
BC00380=237569,209073,1075139
BC00381=238807,208321,1075139
BC00382=238807,208321,1075139
BC00383=238807,208321,1075139
BC00384=223366,211989,1075139
BC00385=221836,212741,1075139
BC00386=241499,229228,1075139
BC00387=320599,204052,1075139
BC00388=360063,167590,1075139
BC00389=355335,166592,1075139
BC00390=353445,166194,1075138
BC00391=353444,166193,1075139
BC00392=353444,166193,1075139
BC00393=356944,167983,1075139
BC00394=359435,168688,1075139
BC00395=364163,169685,1075139
BC00396=364163,169685,1075139
BC00397=304591,281793,1075139
BC00398=304591,281793,1075139
BC00399=288600,338238,1075139
BC00400=288600,338238,1075139
BC00401=304591,281793,1075139
BC00402=304591,281793,1075139
BC00403=231963,309860,1075136
BC00404=231963,309860,1075136
BC00405=233647,324920,1075139
BC00406=233647,324920,1075139
BC00407=231963,309860,1075136
BC00408=231963,309860,1075136
BC00409=231963,309860,1075136
BC00410=326578,332685,1075193
BC00411=323120,336307,1075193
BC00412=321736,337755,1075193
BC00413=321736,337755,1075193
BC00414=321736,337755,1075193
BC00415=328068,340093,1075193
BC00416=323263,322445,1075193
BC00417=321770,322623,1075193
BC00418=322390,320758,1075193
BC00419=323941,316095,1075193
BC00420=233820,289078,1075136
BC00421=238694,234539,1075139
BC00422=239368,211919,1075139
BC00423=219707,213290,1075139
BC00424=222158,212700,1075139
BC00425=219409,211365,1075139
BC00426=219409,211365,1075139
BC00427=222158,212700,1075139
BC00428=223658,211558,1075139
BC00429=224081,211236,1075139
BC00430=242033,210741,1075139
BC00431=246705,210612,1075139
BC00432=247003,212537,1075139
BC00433=247748,217349,1075139
BC00434=209118,260791,1075139
BC00435=202120,268661,1075139
BC00436=139973,338551,1075139
BC00437=139973,338551,1075139
BC00438=139973,338551,1075139
BC00439=139973,338551,1075139
BC00440=139973,338551,1075139
BC00441=139973,338551,1075139
BC00442=139973,338551,1075139
BC00443=139973,338551,1075139
BC00444=212566,287975,1075139
BC00445=254728,263853,1075139
BC00446=341527,214194,1075139
BC00447=346109,215748,1075139
BC00448=346318,212780,1075139
BC00449=346318,212780,1075139
BC00450=346318,212780,1075139
BC00451=364169,223218,1075139
BC00452=354888,219000,1075139
BC00453=391846,222999,1075135
BC00454=398158,226235,1075139
BC00455=310307,229731,1075139
BC00456=299999,233020,1075139
BC00457=301954,231820,1075139
BC00458=302223,231655,1075139
BC00459=302223,231655,1075139
BC00460=309588,229407,1075139
BC00461=307542,230755,1075139
BC00462=302427,234123,1075139
BC00463=333823,236884,1075139
BC00464=361923,239355,1075139
BC00465=359457,233910,1075139
BC00466=358640,232105,1075139
BC00467=358471,231732,1075139
BC00468=358471,231732,1075139
BC00469=358640,232105,1075139
BC00470=358640,232105,1075139
BC00471=361923,284669,1073914
BC00472=121205,299272,1075139
BC00473=121205,232638,1075139
BC00474=121205,232638,1075139
BC00475=120716,231531,1075136
BC00476=120715,231530,1075139
BC00477=120715,231530,1075139
BC00478=65825,241039,1075139
BC00479=65825,241039,1075139
BC00480=66315,266195,1075139
BC00481=148903,446070,1075139
BC00482=196573,468404,1075139
BC00483=204883,494729,820550
BC00484=194359,497622,359020
BC00485=192453,463622,275417
BC00486=190116,421937,172916
BC00487=190116,421937,172916
BC00488=190116,421937,172916
BC00489=190116,421937,172916
BC00490=190116,421937,172916
BC00491=190116,421937,172916
BC00492=190116,421937,172916
BC00493=190116,421937,172916
BC00494=190116,421937,172916
BC00495=190116,421937,172916
BC00496=151318,421937,172916
BC00497=151318,421937,172916
BC00498=151318,421937,172916
BC00499=151318,421937,172916
BC00500=151318,421937,172916
BC00501=151318,421937,172916
BC00502=151318,421937,172916
BC00503=151318,421937,172916
BC00504=151318,421937,172916
BC00505=151318,421937,172916
BC00506=151318,421937,172916
BC00507=151318,421937,172916
BC00508=195439,421937,172916
BC00509=195439,421937,172916
BC00510=227909,421937,172916
BC00511=217404,404822,172916
BC00512=217404,385751,172916
BC00513=217404,385751,172916
BC00514=218620,386619,170840
BC00515=218620,386619,170840
BC00516=218620,386619,170840
BC00517=218620,386619,170840
BC00518=218620,386619,170840
BC00519=218620,386619,170840
BC00520=218620,386619,170840
BC00521=218620,386619,170840
BC00522=218620,386619,170840
BC00523=218620,386619,170840
BC00524=218620,386619,170840
BC00525=218620,386619,170840
BC00526=218620,386619,170840
BC00527=218620,386619,170840
BC00528=218620,386619,170840
BC00529=218620,386619,170840
BC00530=218620,386619,170840
BC00531=218620,386619,170840
BC00532=218620,386619,170840
BC00533=368937,386619,170840
BC00534=368937,386619,423431
BC00535=368937,386619,274402
BC00536=346754,384388,162495
BC00537=366650,381560,260482
BC00538=342198,363507,260482
BC00539=342198,363507,260482
BC00540=342198,363507,260482
BC00541=342198,363507,260482
BC00542=342198,363507,260482
BC00543=342198,363507,260482
BC00544=342198,363507,260482
BC00545=342314,361510,17
BC00546=342314,361510,17
BC00547=342198,363507,260482
BC00548=342198,363507,260482
BC00549=342198,363507,260482
BC00550=323894,437815,291159
BC00551=305901,488791,357451
BC00552=249656,512406,34596
BC00553=237183,418851,142396
BC00554=237183,418851,142396
BC00555=237183,418851,142396
BC00556=237183,418851,120359
BC00557=237184,418850,219439
BC00558=237184,418850,219439
BC00559=237183,418851,120359
BC00560=237183,418851,120359
BC00561=237183,418851,120359
BC00562=251463,428144,17
BC00563=251463,428144,17
BC00564=251463,428144,17
BC00565=251463,428144,17
BC00566=251463,428144,17
BC00567=251463,428144,17
BC00568=251463,428144,17
BC00569=241841,446326,27137
BC00570=220903,485888,86147
BC00571=190116,512106,172916
BC00572=390901,511303,172916
BC00573=353841,494829,153659
BC00574=316410,423960,299876
BC00575=301707,375048,330746
BC00576=301707,375048,330746
BC00577=284369,368690,17
BC00578=284369,368690,17
BC00579=301707,375048,330746
BC00580=301707,375048,330746
BC00581=301707,375048,330746
BC00582=298906,384691,452116
BC00583=261578,485555,421935
BC00584=252426,507061,35762
BC00585=190116,509597,172916
BC00586=239472,457451,34109
BC00587=239472,457451,34109
BC00588=239472,457451,34109
BC00589=251597,466175,17
BC00590=251597,466175,17
BC00591=239472,457451,34109
BC00592=239472,457451,34109
BC00593=232097,459370,27765
BC00594=232097,459370,27765
BC00595=199838,467766,17
BC00596=199838,467766,17
BC00597=232097,459370,27765
BC00598=232097,459370,27765
BC00599=232097,459370,27765
BC00600=219873,484030,70030
BC00601=190116,502733,172916
BC00602=333027,509528,372084
BC00603=325624,426372,445048
BC00604=325269,368711,432113
BC00605=325269,352273,432113
BC00606=313691,388554,17
BC00607=313691,388554,17
BC00608=325269,352273,432113
BC00609=325269,352273,432113
BC00610=325269,361687,432113
BC00611=325269,361687,432113
BC00612=334073,353839,365053
BC00613=334073,353839,365053
BC00614=334073,353839,365053
BC00615=381995,362872,17
BC00616=381995,362872,17
BC00617=334073,353839,365053
BC00618=334073,353839,365053
BC00619=334073,353839,365053
BC00620=334073,353839,365051
BC00621=334073,353839,365051
BC00622=334986,360422,17
BC00623=334986,360422,17
BC00624=334073,353839,365051
BC00625=334073,353839,365051
BC00626=334073,353839,365051
BC00627=334073,353839,365051
BC00628=334073,353839,365051
BC00629=365410,393202,17
BC00630=365410,393202,17
BC00631=334073,353839,365051
BC00632=334073,353839,365051
BC00633=327689,349961,365051
BC00634=327689,349961,365051
BC00635=327689,349961,365051
BC00636=327689,349961,365051
BC00637=327689,349961,365051
BC00638=327689,349961,365051
BC00639=327689,349961,365051
BC00640=365634,399650,17
BC00641=365634,399650,17
BC00642=327689,349961,365051
BC00643=327689,349961,396904
BC00644=398015,435700,359686
BC00645=398015,559674,359686
BC00646=98527,515267,14
BC00647=98527,515267,14
BC00648=164584,515267,14
BC00649=164584,515267,14
BC00650=164584,515267,14
BC00651=164584,515267,14
BC00652=164584,515267,14
BC00653=164584,515267,12
BC00654=164584,515267,12
BC00655=164584,515267,12
BC00656=164584,490178,12
BC00657=164584,490178,12
BC00658=164584,490178,12
BC00659=164584,490178,12
BC00660=164584,490178,12
BC00661=164584,490178,12
BC00662=279707,501261,17
EC00000=-797528,-182698
EC00001=-797528,-182698
EC00002=-798156,-183832
EC00003=-798156,-183832
EC00004=-798156,-183832
EC00005=-798156,-183832
EC00006=-798156,-183832
EC00007=-798156,-183832
EC00008=-798156,-183832
EC00009=-798156,-183832
EC00010=-798155,-183832
EC00011=-798155,-183832
EC00012=-798155,-183832
EC00013=-798155,-183832
EC00014=-798155,-183832
EC00015=-798156,-183832
EC00016=-798156,-183832
EC00017=-798156,-183832
EC00018=-798156,-183832
EC00019=-798156,-183832
EC00020=-798156,-183832
EC00021=-798156,-183832
EC00022=-798156,-183832
EC00023=-798156,-183832
EC00024=-798156,-183832
EC00025=-798156,-183832
EC00026=-798156,-183832
EC00027=-798156,-183832
EC00028=-798156,-183832
EC00029=-798156,-183832
EC00030=-798156,-183832
EC00031=-798156,-183832
EC00032=-798156,-183832
EC00033=-798156,-183832
EC00034=-798156,-183832
EC00035=-798156,-183832
EC00036=-798156,-183832
EC00037=-798156,-183832
EC00038=-798156,-183832
EC00039=-798156,-183832
EC00040=-798156,-183832
EC00041=-798156,-183832
EC00042=-798156,-183832
EC00043=-798156,-183832
EC00044=-798156,-183832
EC00045=-798156,-183832
EC00046=-798156,-183832
EC00047=-798156,-183832
EC00048=-798156,-183832
EC00049=-798156,-183832
EC00050=-798156,-183832
EC00051=-798156,-183832
EC00052=-798156,-183832
EC00053=-798156,-183832
EC00054=-798155,-183833
EC00055=-798154,-183833
EC00056=-798154,-183833
EC00057=-798154,-183833
EC00058=-798154,-183833
EC00059=-798154,-183833
EC00060=-798154,-183833
EC00061=-798154,-183833
EC00062=-798154,-183833
EC00063=-798154,-183833
EC00064=-798154,-183833
EC00065=-798154,-183833
EC00066=-798154,-183833
EC00067=-798154,-183833
EC00068=-798154,-183833
EC00069=-798154,-183833
EC00070=-798154,-183833
EC00071=-798154,-183833
EC00072=-798154,-183833
EC00073=-798154,-183833
EC00074=-798154,-183833
EC00075=-798154,-183833
EC00076=-798154,-183833
EC00077=-798154,-183833
EC00078=-798154,-183833
EC00079=-798154,-183833
EC00080=-798154,-183833
EC00081=-798154,-183833
EC00082=-798154,-183833
EC00083=-798154,-183833
EC00084=-798153,-183833
EC00085=-798153,-183833
EC00086=-798153,-183833
EC00087=-798153,-183833
EC00088=-798154,-183834
EC00089=-798153,-183834
EC00090=-798153,-183834
EC00091=-798153,-183834
EC00092=-798153,-183834
EC00093=-798153,-183834
EC00094=-798153,-183834
EC00095=-798153,-183834
EC00096=-798153,-183834
EC00097=-798153,-183834
EC00098=-798153,-183834
EC00099=-798153,-183834
EC00100=-798153,-183834
EC00101=-798153,-183834
EC00102=-798153,-183834
EC00103=-798153,-183834
EC00104=-798155,-183833
EC00105=-798156,-183832
EC00106=-798156,-183832
EC00107=-798156,-183832
EC00108=-798156,-183832
EC00109=-798156,-183832
EC00110=-798156,-183832
EC00111=-798156,-183832
EC00112=-798156,-183832
EC00113=-798156,-183832
EC00114=-798156,-183832
EC00115=-798156,-183832
EC00116=-798154,-183832
EC00117=-798154,-183832
EC00118=-798154,-183832
EC00119=-798154,-183832
EC00120=-798154,-183832
EC00121=-798156,-183832
EC00122=-798156,-183832
EC00123=-798156,-183832
EC00124=-798156,-183832
EC00125=-798156,-183832
EC00126=-798156,-183832
EC00127=-798156,-183832
EC00128=-798156,-183832
EC00129=-798156,-183832
EC00130=-798156,-183832
EC00131=-798156,-183832
EC00132=-798156,-183832
EC00133=-798156,-183832
EC00134=-798156,-183832
EC00135=-798156,-183832
EC00136=-798156,-183832
EC00137=-798156,-183832
EC00138=-798156,-183832
EC00139=-798156,-183832
EC00140=-798156,-183832
EC00141=-798156,-183832
EC00142=-798156,-183832
EC00143=-798156,-183832
EC00144=-798156,-183832
EC00145=-798156,-183832
EC00146=-798156,-183832
EC00147=-798156,-183832
EC00148=-798156,-183832
EC00149=-798156,-183832
EC00150=-798156,-183832
EC00151=-798156,-183832
EC00152=-798156,-183832
EC00153=-798156,-183832
EC00154=-798156,-183832
EC00155=-798156,-183832
EC00156=-798156,-183832
EC00157=-798156,-183832
EC00158=-798155,-183832
EC00159=-798156,-183832
EC00160=-798156,-183832
EC00161=-798156,-183832
EC00162=-798156,-183832
EC00163=-798156,-183832
EC00164=-798156,-183832
EC00165=-798156,-183832
EC00166=-798156,-183832
EC00167=-798156,-183832
EC00168=-798156,-183832
EC00169=-798156,-183832
EC00170=-798156,-183832
EC00171=-798156,-183832
EC00172=-798156,-183832
EC00173=-798156,-183832
EC00174=-798156,-183832
EC00175=-798156,-183832
EC00176=-798156,-183832
EC00177=-798156,-183832
EC00178=-798156,-183832
EC00179=-798156,-183832
EC00180=-798156,-183832
EC00181=-798156,-183832
EC00182=-798156,-183832
EC00183=-798156,-183832
EC00184=-798156,-183832
EC00185=-798156,-183832
EC00186=-798156,-183832
EC00187=-798156,-183832
EC00188=-798156,-183832
EC00189=-798156,-183832
EC00190=-798156,-183832
EC00191=-798156,-183832
EC00192=-798156,-183832
EC00193=-798156,-183832
EC00194=-798156,-183832
EC00195=-798156,-183832
EC00196=-798156,-183832
EC00197=-798156,-183832
EC00198=-798156,-183832
EC00199=-798156,-183832
EC00200=-798156,-183832
EC00201=-798156,-183832
EC00202=-798156,-183832
EC00203=-798156,-183832
EC00204=-798156,-183832
EC00205=-798156,-183832
EC00206=-798156,-183832
EC00207=-798156,-183832
EC00208=-798156,-183832
EC00209=-798156,-183832
EC00210=-798156,-183832
EC00211=-798156,-183832
EC00212=-798156,-183832
EC00213=-798156,-183832
EC00214=-798156,-183832
EC00215=-798156,-183832
EC00216=-798156,-183832
EC00217=-798156,-183832
EC00218=-798156,-183832
EC00219=-798156,-183832
EC00220=-798156,-183832
EC00221=-798156,-183832
EC00222=-798156,-183832
EC00223=-798156,-183832
EC00224=-798156,-183832
EC00225=-798156,-183832
EC00226=-798156,-183832
EC00227=-798156,-183832
EC00228=-798156,-183832
EC00229=-798156,-183832
EC00230=-798156,-183832
EC00231=-798156,-183832
EC00232=-798156,-183832
EC00233=-798156,-183832
EC00234=-798156,-183832
EC00235=-798155,-183832
EC00236=-798155,-183832
EC00237=-798155,-183832
EC00238=-798155,-183832
EC00239=-798155,-183832
EC00240=-798155,-183832
EC00241=-798155,-183832
EC00242=-798155,-183832
EC00243=-798155,-183832
EC00244=-798155,-183832
EC00245=-798155,-183832
EC00246=-798155,-183832
EC00247=-798155,-183832
EC00248=-798155,-183832
EC00249=-798155,-183832
EC00250=-798155,-183832
EC00251=-798155,-183832
EC00252=-798155,-183832
EC00253=-798155,-183832
EC00254=-798155,-183832
EC00255=-798155,-183832
EC00256=-798155,-183832
EC00257=-798155,-183832
EC00258=-798156,-183832
EC00259=-798156,-183832
EC00260=-798156,-183832
EC00261=-798155,-183833
EC00262=-798156,-183832
EC00263=-798156,-183832
EC00264=-798156,-183832
EC00265=-798156,-183832
EC00266=-798156,-183832
EC00267=-798156,-183832
EC00268=-798156,-183832
EC00269=-798156,-183832
EC00270=-798156,-183832
EC00271=-798156,-183832
EC00272=-798156,-183832
EC00273=-798156,-183832
EC00274=-798156,-183832
EC00275=-798156,-183832
EC00276=-798156,-183832
EC00277=-798156,-183832
EC00278=-798156,-183832
EC00279=-798156,-183832
EC00280=-798155,-183834
EC00281=-975524,-183832
EC00282=-975524,-183832
EC00283=-798156,-183832
EC00284=-798156,-183832
EC00285=-798156,-183832
EC00286=-798156,-183832
EC00287=-975524,-183832
EC00288=-975524,-183832
EC00289=-798156,-183832
EC00290=-798156,-183832
EC00291=-798156,-183832
EC00292=-975524,-183832
EC00293=-975524,-183832
EC00294=-798156,-183832
EC00295=-798156,-183832
EC00296=-798156,-183832
EC00297=-798156,-183832
EC00298=-798155,-183835
EC00299=-975524,-183832
EC00300=-975524,-183832
EC00301=-798156,-183832
EC00302=-798156,-183832
EC00303=-798156,-183832
EC00304=-798156,-183832
EC00305=-798156,-183832
EC00306=-798156,-183832
EC00307=-798156,-183832
EC00308=-798156,-183832
EC00309=-975524,-183832
EC00310=-975524,-183832
EC00311=-798156,-183832
EC00312=-798156,-183832
EC00313=-798156,-183832
EC00314=-798156,-183832
EC00315=-798156,-183832
EC00316=-798156,-183832
EC00317=-798156,-183832
EC00318=-798156,-183832
EC00319=-798156,-183832
EC00320=-798156,-183832
EC00321=-798156,-183832
EC00322=-798156,-183832
EC00323=-798156,-183832
EC00324=-798156,-183832
EC00325=-798156,-183832
EC00326=-798156,-183832
EC00327=-798156,-183832
EC00328=-798156,-183832
EC00329=-798155,-183832
EC00330=-798155,-183832
EC00331=-798156,-183832
EC00332=-798156,-183832
EC00333=-798156,-183832
EC00334=-798156,-183832
EC00335=-798156,-183832
EC00336=-798156,-183832
EC00337=-798156,-183832
EC00338=-798156,-183832
EC00339=-798156,-183832
EC00340=-798156,-183832
EC00341=-798156,-183832
EC00342=-798156,-183832
EC00343=-798156,-183832
EC00344=-798156,-183832
EC00345=-798156,-183832
EC00346=-798156,-183832
EC00347=-798156,-183832
EC00348=-798156,-183832
EC00349=-798156,-183832
EC00350=-798156,-183832
EC00351=-798156,-183832
EC00352=-798156,-183832
EC00353=-798156,-183832
EC00354=-798156,-183832
EC00355=-798156,-183832
EC00356=-798156,-183832
EC00357=-798156,-183832
EC00358=-798156,-183832
EC00359=-798156,-183832
EC00360=-798156,-183832
EC00361=-798156,-183832
EC00362=-798156,-183832
EC00363=-798156,-183832
EC00364=-798156,-183832
EC00365=-798156,-183832
EC00366=-798156,-183832
EC00367=-798156,-183832
EC00368=-798156,-183832
EC00369=-798156,-183832
EC00370=-798156,-183832
EC00371=-798156,-183832
EC00372=-798156,-183832
EC00373=-798156,-183832
EC00374=-798156,-183832
EC00375=-798156,-183832
EC00376=-798156,-183832
EC00377=-798156,-183832
EC00378=-798156,-183832
EC00379=-798156,-183832
EC00380=-798156,-183832
EC00381=-798156,-183832
EC00382=-798156,-183832
EC00383=-798156,-183832
EC00384=-798156,-183832
EC00385=-798156,-183832
EC00386=-798156,-183832
EC00387=-798156,-183832
EC00388=-798156,-183832
EC00389=-798156,-183832
EC00390=-798154,-183835
EC00391=-798156,-183832
EC00392=-798156,-183832
EC00393=-798156,-183832
EC00394=-798156,-183832
EC00395=-798156,-183832
EC00396=-798156,-183832
EC00397=-798156,-183832
EC00398=-798156,-183832
EC00399=-975524,-183832
EC00400=-975524,-183832
EC00401=-798156,-183832
EC00402=-798156,-183832
EC00403=-798154,-183833
EC00404=-798154,-183833
EC00405=-975524,-183832
EC00406=-975524,-183832
EC00407=-798154,-183833
EC00408=-798154,-183833
EC00409=-798154,-183833
EC00410=-975524,-183832
EC00411=-975524,-183832
EC00412=-975524,-183832
EC00413=-975524,-183832
EC00414=-975524,-183832
EC00415=-975524,-183832
EC00416=-975524,-183832
EC00417=-975524,-183832
EC00418=-975524,-183832
EC00419=-975524,-183832
EC00420=-798670,-183833
EC00421=-800023,-183832
EC00422=-798156,-183832
EC00423=-798156,-183832
EC00424=-798156,-183832
EC00425=-798156,-183832
EC00426=-798156,-183832
EC00427=-798156,-183832
EC00428=-798156,-183832
EC00429=-798156,-183832
EC00430=-798156,-183832
EC00431=-798156,-183832
EC00432=-798156,-183832
EC00433=-798156,-183832
EC00434=-798156,-183832
EC00435=-798156,-183832
EC00436=-798156,-183832
EC00437=-798156,-183832
EC00438=-798156,-183832
EC00439=-798156,-183832
EC00440=-798156,-183832
EC00441=-798156,-183832
EC00442=-798156,-183832
EC00443=-798156,-183832
EC00444=-798156,-183832
EC00445=-798156,-183832
EC00446=-798156,-183832
EC00447=-798156,-183832
EC00448=-798156,-183832
EC00449=-798156,-183832
EC00450=-798156,-183832
EC00451=-798156,-183832
EC00452=-798156,-183832
EC00453=-798155,-183832
EC00454=-798156,-183832
EC00455=-798156,-183832
EC00456=-798156,-183832
EC00457=-798156,-183832
EC00458=-798156,-183832
EC00459=-798156,-183832
EC00460=-798156,-183832
EC00461=-798156,-183832
EC00462=-798156,-183832
EC00463=-798156,-183832
EC00464=-798156,-183832
EC00465=-798156,-183832
EC00466=-798156,-183832
EC00467=-798156,-183832
EC00468=-798156,-183832
EC00469=-798156,-183832
EC00470=-798156,-183832
EC00471=-798156,-183832
EC00472=-798156,-183832
EC00473=-798156,-183832
EC00474=-798156,-183832
EC00475=-798154,-183832
EC00476=-798156,-183832
EC00477=-798156,-183832
EC00478=-798156,-183832
EC00479=-798156,-183832
EC00480=-798156,-183832
EC00481=-798156,-183832
EC00482=-798156,-183832
EC00483=-798156,-183832
EC00484=-798156,-183832
EC00485=-798156,-183832
EC00486=-798156,-183832
EC00487=-798156,-183832
EC00488=-798156,-183832
EC00489=-798156,-183832
EC00490=-798156,-183832
EC00491=-798156,-183832
EC00492=-798156,-183832
EC00493=-798156,-183832
EC00494=-798156,-183832
EC00495=-798156,-183832
EC00496=-798156,-183832
EC00497=-798156,-183832
EC00498=-798156,-183832
EC00499=-798156,-183832
EC00500=-798156,-183832
EC00501=-798156,-183832
EC00502=-798156,-183832
EC00503=-798156,-183832
EC00504=-798156,-183832
EC00505=-798156,-183832
EC00506=-798156,-183832
EC00507=-798156,-183832
EC00508=-798156,-183832
EC00509=-798156,-183832
EC00510=-798156,-183832
EC00511=-798156,-183832
EC00512=-798156,-183832
EC00513=-798156,-183832
EC00514=-798155,-183833
EC00515=-798155,-183833
EC00516=-798155,-183833
EC00517=-798155,-183833
EC00518=-798155,-183833
EC00519=-798155,-183833
EC00520=-798155,-183833
EC00521=-798155,-183833
EC00522=-798155,-183833
EC00523=-798155,-183833
EC00524=-798155,-183833
EC00525=-798155,-183833
EC00526=-798155,-183833
EC00527=-798155,-183833
EC00528=-798155,-183833
EC00529=-798155,-183833
EC00530=-798155,-183833
EC00531=-798155,-183833
EC00532=-798155,-183833
EC00533=-798155,-183833
EC00534=-798155,-183833
EC00535=-798155,-183833
EC00536=-798155,-183833
EC00537=-798156,-183832
EC00538=-798156,-183832
EC00539=-798156,-183832
EC00540=-798156,-183832
EC00541=-798156,-183832
EC00542=-798156,-183832
EC00543=-798156,-183832
EC00544=-798156,-183832
EC00545=-798156,-183832
EC00546=-798156,-183832
EC00547=-798156,-183832
EC00548=-798156,-183832
EC00549=-798156,-183832
EC00550=-798155,-183833
EC00551=-798155,-183833
EC00552=-798155,-183833
EC00553=-798154,-183832
EC00554=-798154,-183832
EC00555=-798154,-183832
EC00556=-798154,-183832
EC00557=-798156,-183832
EC00558=-798156,-183832
EC00559=-798154,-183832
EC00560=-798154,-183832
EC00561=-798154,-183832
EC00562=-798156,-183832
EC00563=-798156,-183832
EC00564=-798156,-183832
EC00565=-798156,-183832
EC00566=-798156,-183832
EC00567=-798156,-183832
EC00568=-798156,-183832
EC00569=-798156,-183832
EC00570=-798156,-183832
EC00571=-798156,-183832
EC00572=-798156,-183832
EC00573=-798156,-183832
EC00574=-798156,-183832
EC00575=-798156,-183832
EC00576=-798156,-183832
EC00577=-798156,-183832
EC00578=-798156,-183832
EC00579=-798156,-183832
EC00580=-798156,-183832
EC00581=-798156,-183832
EC00582=-798156,-183832
EC00583=-798156,-183832
EC00584=-798156,-183832
EC00585=-798156,-183832
EC00586=-798154,-183832
EC00587=-798154,-183832
EC00588=-798154,-183832
EC00589=-798156,-183832
EC00590=-798156,-183832
EC00591=-798154,-183832
EC00592=-798154,-183832
EC00593=-798154,-183832
EC00594=-798154,-183832
EC00595=-798156,-183832
EC00596=-798156,-183832
EC00597=-798154,-183832
EC00598=-798154,-183832
EC00599=-798154,-183832
EC00600=-798155,-183832
EC00601=-798156,-183832
EC00602=-798156,-183832
EC00603=-798156,-183832
EC00604=-798156,-183832
EC00605=-798156,-183832
EC00606=-798156,-183832
EC00607=-798156,-183832
EC00608=-798156,-183832
EC00609=-798156,-183832
EC00610=-798156,-183832
EC00611=-798156,-183832
EC00612=-798156,-183832
EC00613=-798156,-183832
EC00614=-798156,-183832
EC00615=-798156,-183832
EC00616=-798156,-183832
EC00617=-798156,-183832
EC00618=-798156,-183832
EC00619=-798156,-183832
EC00620=-798156,-183832
EC00621=-798156,-183832
EC00622=-798156,-183832
EC00623=-798156,-183832
EC00624=-798156,-183832
EC00625=-798156,-183832
EC00626=-798156,-183832
EC00627=-798156,-183832
EC00628=-798156,-183832
EC00629=-798156,-183832
EC00630=-798156,-183832
EC00631=-798156,-183832
EC00632=-798156,-183832
EC00633=-798156,-183832
EC00634=-798156,-183832
EC00635=-798156,-183832
EC00636=-798156,-183832
EC00637=-798156,-183832
EC00638=-798156,-183832
EC00639=-798156,-183832
EC00640=-798156,-183832
EC00641=-798156,-183832
EC00642=-798156,-183832
EC00643=-798156,-183832
EC00644=-798156,-183832
EC00645=-798156,-183832
EC00646=-798155,-183833
EC00647=-798155,-183833
EC00648=-798155,-183833
EC00649=-798155,-183833
EC00650=-798155,-183833
EC00651=-798155,-183833
EC00652=-798155,-183833
EC00653=-798153,-183833
EC00654=-798153,-183833
EC00655=-798153,-183833
EC00656=-798153,-183833
EC00657=-798153,-183833
EC00658=-798153,-183833
EC00659=-798153,-183833
EC00660=-798153,-183833
EC00661=-798153,-183833
EC00662=-798156,-183832
///POSTYPE BASE
///RECTAN
///RCONF 0,0,0,0,1,0,0,0,0,0,0,0,0,0,0,0,0,0,0,0,0,0,0,0
P00006=2.006,1.622,-0.565,0.0000,0.0000,0.0000
P00021=0.073,2.058,-0.109,0.0000,0.0000,0.0000
P00022=2.006,1.622,-0.565,0.0000,0.0000,0.0000
///RCONF 0,0,0,0,0,0,0,0,0,0,0,0,0,0,0,0,0,0,0,0,0,0,0,0
P00023=-2.957,-4.083,2.762,0.0000,0.0000,0.0000
P00030=-0.014,-0.768,0.131,0.0000,0.0000,0.0000
P00031=-0.170,0.039,-0.647,0.0000,0.0000,0.0000
P00032=-0.423,0.157,3.222,0.0000,0.0000,0.0000
P00033=0.854,-1.099,3.047,0.0000,0.0000,0.0000
///RCONF 0,0,0,0,1,0,0,0,0,0,0,0,0,0,0,0,0,0,0,0,0,0,0,0
P00034=-8.151,9.743,-4.393,0.0000,0.0000,0.0000
///RCONF 0,0,0,0,0,0,0,0,0,0,0,0,0,0,0,0,0,0,0,0,0,0,0,0
P00035=0.390,-0.027,1.040,0.0000,0.0000,0.0000
P00036=-2.434,0.084,0.197,0.0000,0.0000,0.0000
P00037=-1.075,5.090,-3.949,0.0000,0.0000,0.0000
P00038=0.174,-1.527,-10.860,0.0000,0.0000,0.0000
P00039=-0.109,1.838,-0.266,0.0000,0.0000,0.0000
P00040=2.716,-0.016,3.014,0.0000,0.0000,0.0000
P00041=-0.109,0.014,0.966,0.0000,0.0000,0.0000
P00042=-0.220,0.371,-0.613,0.0000,0.0000,0.0000
P00050=-0.123,2.174,-1.314,0.0000,0.0000,0.0000
P00052=-0.153,5.586,-7.982,0.0000,0.0000,0.0000
P00055=-0.009,2.790,-4.790,0.0000,0.0000,0.0000
P00056=3.147,0.012,0.038,0.0000,0.0000,0.0000
P00057=13.307,-11.525,-2.645,0.0000,0.0000,0.0000
P00058=6.894,-13.094,-1.754,0.0000,0.0000,0.0000
P00060=1524.284,698.404,-261.973,-0.4635,36.8346,-1.2388
P00090=-14.057,13.261,-6.464,0.0000,0.0000,0.0000
P00091=1.048,0.648,3.624,0.0000,0.0000,0.0000
//INST
///DATE 2024/11/25 13:36
///ATTR SC,RW
///GROUP1 RB1,BS1
///GROUP2 ST1
NOP
'OK_r2_O8A-O21A(90,0)
'Path S1018
MOVJ C00000 BC00000 VJ=50.00  +MOVJ EC00000 VJ=10.00
MOVJ C00001 BC00001 VJ=100.00  +MOVJ EC00001 VJ=100.00
SFTOF3D
MOVJ C00002 BC00002 VJ=100.00  +MOVJ EC00002 VJ=100.00
MOVL C00003 BC00003 V=400.0  +MOVJ EC00003 VJ=100.00
SMOVL C00004 BC00004 V=100.0  +MOVJ EC00004
SREFP 3 C00005 BC00005  +REFP EC00005
CALL JOB:SEARCH-R1-S13D
SET P031 P006
SFTON3D P031
SMOVL C00006 BC00006 V=100.0  +MOVJ EC00006
SREFP 3 C00007 BC00007  +REFP EC00007
CALL JOB:SEARCH-R1-S13D
SET P031 P006
SFTON3D P031
SFTOF3D
SMOVL C00008 BC00008 V=100.0  +MOVJ EC00008
MOVL C00009 BC00009 V=333.3  +MOVJ EC00009 VJ=100.00
SMOVL C00010 BC00010 V=100.0  +MOVJ EC00010
SREFP 3 C00011 BC00011  +REFP EC00011
CALL JOB:SEARCH-R1-S13D
SET P032 P006
SFTON3D P032
SMOVL C00012 BC00012 V=100.0  +MOVJ EC00012
SREFP 3 C00013 BC00013  +REFP EC00013
CALL JOB:SEARCH-R1-S13D
SET P032 P006
SFTON3D P032
SMOVL C00014 BC00014 V=250.0  +MOVJ EC00014
MOVL C00015 BC00015 V=1000.0  +MOVJ EC00015 VJ=100.00
'Path S1554
SFTOF3D
MOVJ C00016 BC00016 VJ=100.00  +MOVJ EC00016 VJ=100.00
MOVL C00017 BC00017 V=400.0  +MOVJ EC00017 VJ=100.00
SMOVL C00018 BC00018 V=100.0  +MOVJ EC00018
SMOVL C00019 BC00019 V=100.0  +MOVJ EC00019
SREFP 3 C00020 BC00020  +REFP EC00020
CALL JOB:SEARCH-R1-S13D
SET P035 P006
SFTON3D P035
SMOVL C00021 BC00021 V=100.0  +MOVJ EC00021
SMOVL C00022 BC00022 V=100.0  +MOVJ EC00022
SMOVL C00023 BC00023 V=100.0  +MOVJ EC00023
SREFP 3 C00024 BC00024  +REFP EC00024
CALL JOB:SEARCH-R1-S13D
SET P035 P006
SFTON3D P035
SMOVL C00025 BC00025 V=166.7  +MOVJ EC00025
MOVL C00026 BC00026 V=1000.0  +MOVJ EC00026 VJ=100.00
MOVJ C00027 BC00027 VJ=50.00  +MOVJ EC00027 VJ=10.00
MOVJ C00028 BC00028 VJ=100.00  +MOVJ EC00028 VJ=100.00
'Path S1019
SFTOF3D
MOVJ C00029 BC00029 VJ=100.00  +MOVJ EC00029 VJ=100.00
MOVL C00030 BC00030 V=400.0  +MOVJ EC00030 VJ=100.00
SMOVL C00031 BC00031 V=100.0  +MOVJ EC00031
SREFP 3 C00032 BC00032  +REFP EC00032
CALL JOB:SEARCH-R1-S13D
SET P050 P006
SFTON3D P050
SMOVL C00033 BC00033 V=100.0  +MOVJ EC00033
SREFP 3 C00034 BC00034  +REFP EC00034
CALL JOB:SEARCH-R1-S13D
SET P050 P006
SFTON3D P050
SMOVL C00035 BC00035 V=166.7  +MOVJ EC00035
SMOVL C00036 BC00036 V=166.7  +MOVJ EC00036
SREFP 3 C00037 BC00037  +REFP EC00037
CALL JOB:SEARCH-R1-S13D
SET P050 P006
SFTON3D P050
SMOVL C00038 BC00038 V=166.7  +MOVJ EC00038
MOVL C00039 BC00039 V=1000.0  +MOVJ EC00039 VJ=100.00
MOVJ C00040 BC00040 VJ=100.00  +MOVJ EC00040 VJ=100.00
'OBROT 110
MOVJ C00041 BC00041 VJ=100.00  +MOVJ EC00041 VJ=100.00
MOVJ C00042 BC00042 VJ=100.00  +MOVJ EC00042 VJ=100.00
MOVJ C00043 BC00043 VJ=100.00  +MOVJ EC00043 VJ=100.00
'Path S1020
SFTOF3D
SMOVL C00044 BC00044 V=166.7  +MOVJ EC00044
SREFP 3 C00045 BC00045  +REFP EC00045
CALL JOB:SEARCH-R1-S13D
SET P033 P006
SFTON3D P033
SMOVL C00046 BC00046 V=166.7  +MOVJ EC00046
SREFP 3 C00047 BC00047  +REFP EC00047
CALL JOB:SEARCH-R1-S13D
SET P033 P006
SFTON3D P033
MOVJ C00048 BC00048 VJ=50.00  +MOVJ EC00048 VJ=50.00
MOVJ C00049 BC00049 VJ=50.00  +MOVJ EC00049 VJ=100.00
SMOVL C00050 BC00050 V=100.0  +MOVJ EC00050
SREFP 3 C00051 BC00051  +REFP EC00051
CALL JOB:SEARCH-R1-S13D
SET P033 P006
SFTON3D P033
SMOVL C00052 BC00052 V=166.7  +MOVJ EC00052
MOVL C00053 BC00053 V=666.7  +MOVJ EC00053 VJ=100.00
MOVJ C00054 BC00054 VJ=50.00  +MOVJ EC00054 VJ=50.00
MOVJ C00055 BC00055 VJ=50.00  +MOVJ EC00055 VJ=50.00
MOVJ C00056 BC00056 VJ=50.00  +MOVJ EC00056 VJ=50.00
'Path S1025
SFTOF3D
SMOVL C00057 BC00057 V=60.0  +MOVJ EC00057
SREFP 3 C00058 BC00058  +REFP EC00058
CALL JOB:SEARCH-R1-S13D
SET P038 P006
SFTON3D P038
SMOVL C00059 BC00059 V=100.0  +MOVJ EC00059
SREFP 3 C00060 BC00060  +REFP EC00060
CALL JOB:SEARCH-R1-S13D
SET P038 P006
SFTON3D P038
SMOVL C00061 BC00061 V=100.0  +MOVJ EC00061
SMOVL C00062 BC00062 V=166.7  +MOVJ EC00062
MOVJ C00063 BC00063 VJ=100.00  +MOVJ EC00063 VJ=15.00
MOVJ C00064 BC00064 VJ=100.00  +MOVJ EC00064 VJ=50.00
MOVJ C00065 BC00065 VJ=100.00  +MOVJ EC00065 VJ=15.00
MOVJ C00066 BC00066 VJ=15.00  +MOVJ EC00066 VJ=50.00
SMOVL C00067 BC00067 V=100.0  +MOVJ EC00067
SREFP 3 C00068 BC00068  +REFP EC00068
CALL JOB:SEARCH-R1-S13D
SET P038 P006
SFTON3D P038
SMOVL C00069 BC00069 V=100.0  +MOVJ EC00069
MOVJ C00070 BC00070 VJ=100.00  +MOVJ EC00070 VJ=15.00
MOVL C00071 BC00071 V=833.3  +MOVJ EC00071 VJ=100.00
MOVJ C00072 BC00072 VJ=100.00  +MOVJ EC00072 VJ=15.00
MOVJ C00073 BC00073 VJ=100.00  +MOVJ EC00073 VJ=15.00
'Path S1027
SFTOF3D
MOVL C00074 BC00074 V=400.0  +MOVJ EC00074 VJ=100.00
SMOVL C00075 BC00075 V=100.0  +MOVJ EC00075
SREFP 3 C00076 BC00076  +REFP EC00076
CALL JOB:SEARCH-R1-S13D
SET P040 P006
SFTON3D P040
SMOVL C00077 BC00077 V=100.0  +MOVJ EC00077
SMOVL C00078 BC00078 V=133.3  +MOVJ EC00078
SMOVL C00079 BC00079 V=100.0  +MOVJ EC00079
SREFP 3 C00080 BC00080  +REFP EC00080
CALL JOB:SEARCH-R1-S13D
SET P040 P006
SFTON3D P040
SMOVL C00081 BC00081 V=133.3  +MOVJ EC00081
MOVJ C00082 BC00082 VJ=100.00  +MOVJ EC00082 VJ=15.00
MOVJ C00083 BC00083 VJ=100.00  +MOVJ EC00083 VJ=15.00
SMOVL C00084 BC00084 V=100.0  +MOVJ EC00084
SREFP 3 C00085 BC00085  +REFP EC00085
CALL JOB:SEARCH-R1-S13D
SET P040 P006
SFTON3D P040
SMOVL C00086 BC00086 V=100.0  +MOVJ EC00086
'Path S1023
SFTOF3D
MOVJ C00087 BC00087 VJ=100.00  +MOVJ EC00087 VJ=15.00
MOVJ C00088 BC00088 VJ=50.00  +MOVJ EC00088 VJ=15.00
MOVJ C00089 BC00089 VJ=50.00  +MOVJ EC00089 VJ=15.00
MOVJ C00090 BC00090 VJ=50.00  +MOVJ EC00090 VJ=15.00
SMOVL C00091 BC00091 V=100.0  +MOVJ EC00091
SREFP 3 C00092 BC00092  +REFP EC00092
CALL JOB:SEARCH-R1-S13D
SET P036 P006
SFTON3D P036
SMOVL C00093 BC00093 V=100.0  +MOVJ EC00093
SREFP 3 C00094 BC00094  +REFP EC00094
CALL JOB:SEARCH-R1-S13D
SET P036 P006
SFTON3D P036
SMOVL C00095 BC00095 V=100.0  +MOVJ EC00095
SMOVL C00096 BC00096 V=133.3  +MOVJ EC00096
SMOVL C00097 BC00097 V=100.0  +MOVJ EC00097
SREFP 3 C00098 BC00098  +REFP EC00098
CALL JOB:SEARCH-R1-S13D
SET P036 P006
SFTON3D P036
SMOVL C00099 BC00099 V=100.0  +MOVJ EC00099
SMOVL C00100 BC00100 V=250.0  +MOVJ EC00100
SMOVL C00101 BC00101 V=833.3  +MOVJ EC00101
MOVJ C00102 BC00102 VJ=100.00  +MOVJ EC00102 VJ=15.00
MOVJ C00103 BC00103 VJ=100.00  +MOVJ EC00103 VJ=15.00
MOVJ C00104 BC00104 VJ=100.00  +MOVJ EC00104 VJ=15.00
'Path S1024
SFTOF3D
MOVJ C00105 BC00105 VJ=100.00  +MOVJ EC00105 VJ=100.00
MOVL C00106 BC00106 V=400.0  +MOVJ EC00106 VJ=100.00
SMOVL C00107 BC00107 V=100.0  +MOVJ EC00107
SREFP 3 C00108 BC00108  +REFP EC00108
CALL JOB:SEARCH-R1-S13D
SET P037 P006
SFTON3D P037
SMOVL C00109 BC00109 V=100.0  +MOVJ EC00109
SREFP 3 C00110 BC00110  +REFP EC00110
CALL JOB:SEARCH-R1-S13D
SET P037 P006
SFTON3D P037
SMOVL C00111 BC00111 V=100.0  +MOVJ EC00111
MOVL C00112 BC00112 V=400.0  +MOVJ EC00112 VJ=100.00
MOVL C00113 BC00113 V=1000.0  +MOVJ EC00113 VJ=100.00
MOVJ C00114 BC00114 VJ=100.00  +MOVJ EC00114 VJ=100.00
'Path S1028
SFTOF3D
MOVJ C00115 BC00115 VJ=100.00  +MOVJ EC00115 VJ=100.00
SMOVL C00116 BC00116 V=100.0  +MOVJ EC00116
SREFP 3 C00117 BC00117  +REFP EC00117
CALL JOB:SEARCH-R1-S13D
SET P041 P006
SFTON3D P041
SMOVL C00118 BC00118 V=100.0  +MOVJ EC00118
SREFP 3 C00119 BC00119  +REFP EC00119
CALL JOB:SEARCH-R1-S13D
SET P041 P006
SFTON3D P041
SFTOF3D
SMOVL C00120 BC00120 V=100.0  +MOVJ EC00120
MOVL C00121 BC00121 V=400.0  +MOVJ EC00121 VJ=100.00
MOVL C00122 BC00122 V=400.0  +MOVJ EC00122 VJ=15.00
SMOVL C00123 BC00123 V=100.0  +MOVJ EC00123
SREFP 3 C00124 BC00124  +REFP EC00124
CALL JOB:SEARCH-R1-S13D
SET P042 P006
SFTON3D P042
SMOVL C00125 BC00125 V=100.0  +MOVJ EC00125
SREFP 3 C00126 BC00126  +REFP EC00126
CALL JOB:SEARCH-R1-S13D
SET P042 P006
SFTON3D P042
SMOVL C00127 BC00127 V=100.0  +MOVJ EC00127
MOVL C00128 BC00128 V=1000.0  +MOVJ EC00128 VJ=100.00
'Path S1029
MOVJ C00129 BC00129 VJ=100.00  +MOVJ EC00129 VJ=10.00
MOVJ C00130 BC00130 VJ=100.00  +MOVJ EC00130 VJ=10.00
SFTOF3D
MOVJ C00131 BC00131 VJ=100.00  +MOVJ EC00131 VJ=100.00
MOVL C00132 BC00132 V=400.0  +MOVJ EC00132 VJ=100.00
SMOVL C00133 BC00133 V=100.0  +MOVJ EC00133
SREFP 3 C00134 BC00134  +REFP EC00134
CALL JOB:SEARCH-R1-S13D
SET P052 P006
SFTON3D P052
SMOVL C00135 BC00135 V=100.0  +MOVJ EC00135
SMOVL C00136 BC00136 V=100.0  +MOVJ EC00136
SREFP 3 C00137 BC00137  +REFP EC00137
CALL JOB:SEARCH-R1-S13D
SET P052 P006
SFTON3D P052
SMOVL C00138 BC00138 V=133.3  +MOVJ EC00138
MOVL C00139 BC00139 V=400.0  +MOVJ EC00139 VJ=100.00
MOVL C00140 BC00140 V=1000.0  +MOVJ EC00140 VJ=100.00
MOVJ C00141 BC00141 VJ=100.00  +MOVJ EC00141 VJ=10.00
MOVJ C00142 BC00142 VJ=100.00  +MOVJ EC00142 VJ=100.00
MOVL C00143 BC00143 V=1000.0  +MOVJ EC00143 VJ=100.00
SMOVL C00144 BC00144 V=500.0  +MOVJ EC00144
SMOVL C00145 BC00145 V=166.7  +MOVJ EC00145
SREFP 3 C00146 BC00146  +REFP EC00146
CALL JOB:SEARCH-R1-S13D
SET P055 P006
SFTON3D P055
SMOVL C00147 BC00147 V=100.0  +MOVJ EC00147
SREFP 3 C00148 BC00148  +REFP EC00148
CALL JOB:SEARCH-R1-S13D
SET P055 P006
SFTON3D P055
SMOVL C00149 BC00149 V=166.7  +MOVJ EC00149
SFTOF3D
SMOVL C00150 BC00150 V=500.0  +MOVJ EC00150
SMOVL C00151 BC00151 V=166.7  +MOVJ EC00151
SREFP 3 C00152 BC00152  +REFP EC00152
CALL JOB:SEARCH-R1-S13D
SET P060 P006
SFTON3D P060
SMOVL C00153 BC00153 V=100.0  +MOVJ EC00153
SREFP 3 C00154 BC00154  +REFP EC00154
CALL JOB:SEARCH-R1-S13D
SET P060 P006
SFTON3D P060
SMOVL C00155 BC00155 V=166.7  +MOVJ EC00155
SMOVL C00156 BC00156 V=666.7  +MOVJ EC00156
MOVJ C00157 BC00157 VJ=100.00  +MOVJ EC00157 VJ=100.00
'Path S1026
SFTOF3D
MOVJ C00158 BC00158 VJ=100.00  +MOVJ EC00158 VJ=10.00
MOVJ C00159 BC00159 VJ=100.00  +MOVJ EC00159 VJ=100.00
MOVL C00160 BC00160 V=400.0  +MOVJ EC00160 VJ=100.00
SMOVL C00161 BC00161 V=166.7  +MOVJ EC00161
SREFP 3 C00162 BC00162  +REFP EC00162
CALL JOB:SEARCH-R1-S13D
SET P039 P006
SFTON3D P039
SMOVL C00163 BC00163 V=100.0  +MOVJ EC00163
SMOVL C00164 BC00164 V=100.0  +MOVJ EC00164
SREFP 3 C00165 BC00165  +REFP EC00165
CALL JOB:SEARCH-R1-S13D
SET P039 P006
SFTON3D P039
SMOVL C00166 BC00166 V=166.7  +MOVJ EC00166
SMOVL C00167 BC00167 V=333.3  +MOVJ EC00167
SMOVL C00168 BC00168 V=100.0  +MOVJ EC00168
SREFP 3 C00169 BC00169  +REFP EC00169
CALL JOB:SEARCH-R1-S13D
SET P039 P006
SFTON3D P039
SMOVL C00170 BC00170 V=100.0  +MOVJ EC00170
SMOVL C00171 BC00171 V=250.0  +MOVJ EC00171
SMOVL C00172 BC00172 V=166.7  +MOVJ EC00172
MOVL C00173 BC00173 V=400.0  +MOVJ EC00173 VJ=100.00
MOVL C00174 BC00174 V=1000.0  +MOVJ EC00174 VJ=100.00
'Path S1021
SFTOF3D
MOVJ C00175 BC00175 VJ=100.00  +MOVJ EC00175 VJ=100.00
MOVL C00176 BC00176 V=400.0  +MOVJ EC00176 VJ=100.00
SMOVL C00177 BC00177 V=100.0  +MOVJ EC00177
SREFP 3 C00178 BC00178  +REFP EC00178
CALL JOB:SEARCH-R1-S13D
SET P034 P006
SFTON3D P034
SMOVL C00179 BC00179 V=100.0  +MOVJ EC00179
SMOVL C00180 BC00180 V=133.3  +MOVJ EC00180
SMOVL C00181 BC00181 V=100.0  +MOVJ EC00181
SREFP 3 C00182 BC00182  +REFP EC00182
CALL JOB:SEARCH-R1-S13D
SET P034 P006
SFTON3D P034
SMOVL C00183 BC00183 V=100.0  +MOVJ EC00183
SMOVL C00184 BC00184 V=100.0  +MOVJ EC00184
SREFP 3 C00185 BC00185  +REFP EC00185
CALL JOB:SEARCH-R1-S13D
SET P034 P006
SFTON3D P034
SMOVL C00186 BC00186 V=133.3  +MOVJ EC00186
MOVL C00187 BC00187 V=400.0  +MOVJ EC00187 VJ=100.00
MOVL C00188 BC00188 V=1000.0  +MOVJ EC00188 VJ=100.00
MOVJ C00189 BC00189 VJ=100.00  +MOVJ EC00189 VJ=100.00
MOVJ C00190 BC00190 VJ=100.00  +MOVJ EC00190 VJ=100.00
MOVJ C00191 BC00191 VJ=100.00  +MOVJ EC00191 VJ=100.00
SMOVL C00192 BC00192 V=100.0  +MOVJ EC00192
SREFP 3 C00193 BC00193  +REFP EC00193
CALL JOB:SEARCH-R1-S13D
SET P056 P006
SFTON3D P056
SMOVL C00194 BC00194 V=100.0  +MOVJ EC00194
SREFP 3 C00195 BC00195  +REFP EC00195
CALL JOB:SEARCH-R1-S13D
SET P056 P006
SFTON3D P056
SFTOF3D
SMOVL C00196 BC00196 V=100.0  +MOVJ EC00196
SMOVL C00197 BC00197 V=250.0  +MOVJ EC00197
SMOVL C00198 BC00198 V=100.0  +MOVJ EC00198
SREFP 3 C00199 BC00199  +REFP EC00199
CALL JOB:SEARCH-R1-S13D
SET P057 P006
SFTON3D P057
SMOVL C00200 BC00200 V=100.0  +MOVJ EC00200
SREFP 3 C00201 BC00201  +REFP EC00201
CALL JOB:SEARCH-R1-S13D
SET P057 P006
SFTON3D P057
SFTOF3D
SMOVL C00202 BC00202 V=100.0  +MOVJ EC00202
SMOVL C00203 BC00203 V=333.3  +MOVJ EC00203
MOVJ C00204 BC00204 VJ=100.00  +MOVJ EC00204 VJ=100.00
MOVJ C00205 BC00205 VJ=100.00  +MOVJ EC00205 VJ=100.00
MOVJ C00206 BC00206 VJ=100.00  +MOVJ EC00206 VJ=100.00
SMOVL C00207 BC00207 V=166.7  +MOVJ EC00207
SREFP 3 C00208 BC00208  +REFP EC00208
CALL JOB:SEARCH-R1-S13D
SET P058 P006
SFTON3D P058
SMOVL C00209 BC00209 V=166.7  +MOVJ EC00209
SREFP 3 C00210 BC00210  +REFP EC00210
CALL JOB:SEARCH-R1-S13D
SET P058 P006
SFTON3D P058
SFTOF3D
SMOVL C00211 BC00211 V=166.7  +MOVJ EC00211
SMOVL C00212 BC00212 V=666.7  +MOVJ EC00212
MOVJ C00213 BC00213 VJ=100.00  +MOVJ EC00213 VJ=100.00
MOVJ C00214 BC00214 VJ=100.00  +MOVJ EC00214 VJ=100.00
SMOVL C00215 BC00215 V=666.7  +MOVJ EC00215
SMOVL C00216 BC00216 V=166.7  +MOVJ EC00216
SREFP 3 C00217 BC00217  +REFP EC00217
CALL JOB:SEARCH-R1-S13D
SET P090 P006
SFTON3D P090
SMOVL C00218 BC00218 V=166.7  +MOVJ EC00218
SREFP 3 C00219 BC00219  +REFP EC00219
CALL JOB:SEARCH-R1-S13D
SET P090 P006
SFTON3D P090
SFTOF3D
SMOVL C00220 BC00220 V=166.7  +MOVJ EC00220
SMOVL C00221 BC00221 V=500.0  +MOVJ EC00221
SMOVL C00222 BC00222 V=166.7  +MOVJ EC00222
SREFP 3 C00223 BC00223  +REFP EC00223
CALL JOB:SEARCH-R1-S13D
SET P091 P006
SFTON3D P091
SMOVL C00224 BC00224 V=166.7  +MOVJ EC00224
SREFP 3 C00225 BC00225  +REFP EC00225
CALL JOB:SEARCH-R1-S13D
SET P091 P006
SFTON3D P091
SFTOF3D
SMOVL C00226 BC00226 V=166.7  +MOVJ EC00226
MACRO1 MJ#(0) ARGF6
SFTON3D P091
SMOVL C00227 BC00227 V=133.3  +MOVJ EC00227
ARCON
SMOVL C00228 BC00228 V=12.5  +MOVJ EC00228
SFTON3D P090
SMOVL C00229 BC00229 V=12.5  +MOVJ EC00229
ARCOF
SFTOF3D
SMOVL C00230 BC00230 V=166.7  +MOVJ EC00230
SMOVL C00231 BC00231 V=1000.0  +MOVJ EC00231
MOVJ C00232 BC00232 VJ=100.00  +MOVJ EC00232 VJ=100.00
MOVJ C00233 BC00233 VJ=100.00  +MOVJ EC00233 VJ=100.00
MACRO1 MJ#(0) ARGF14
SFTON3D P034
SMOVL C00234 BC00234 V=166.7  +MOVJ EC00234
ARCON
SMOVL C00235 BC00235 V=11.7  +MOVJ EC00235
ARCOF
MOVJ C00236 BC00236 VJ=25.00  +MOVJ EC00236 VJ=100.00
MOVJ C00237 BC00237 VJ=100.00  +MOVJ EC00237 VJ=25.00
SFTON3D P058
SMOVL C00238 BC00238 V=166.7  +MOVJ EC00238
ARCON
SMOVL C00239 BC00239 V=10.0  +MOVJ EC00239
ARCOF
SFTOF3D
SMOVL C00240 BC00240 V=166.7  +MOVJ EC00240
MACRO1 MJ#(0) ARGF9
SMOVL C00241 BC00241 V=500.0  +MOVJ EC00241
SFTON3D P034
SMOVL C00242 BC00242 V=250.0  +MOVJ EC00242
ARCON
SMOVL C00243 BC00243 V=9.2  +MOVJ EC00243
SFTON3D P057
SMOVL C00244 BC00244 V=9.2  +MOVJ EC00244
SMOVL C00245 BC00245 V=9.2  +MOVJ EC00245
SREFP 1 C00246 BC00246  +REFP EC00246
SREFP 2 C00247 BC00247  +REFP EC00247
SFTON3D P056
SWVON WEV#(30)
SMOVL C00248 BC00248 V=8.7  +MOVJ EC00248
SMOVL C00249 BC00249 V=8.7  +MOVJ EC00249
SMOVL C00250 BC00250 V=8.7  +MOVJ EC00250
ARCOF
SWVOF
SFTOF3D
SMOVL C00251 BC00251 V=333.3  +MOVJ EC00251
MOVJ C00252 BC00252 VJ=100.00  +MOVJ EC00252 VJ=25.00
MOVJ C00253 BC00253 VJ=100.00  +MOVJ EC00253 VJ=25.00
SFTON3D P057
SMOVL C00254 BC00254 V=166.7  +MOVJ EC00254
ARCON
SWVON WEV#(30)
SMOVL C00255 BC00255 V=9.2  +MOVJ EC00255
ARCOF
SWVOF
SFTOF3D
SMOVL C00256 BC00256 V=166.7  +MOVJ EC00256
MOVJ C00257 BC00257 VJ=100.00  +MOVJ EC00257 VJ=25.00
'
MOVJ C00258 BC00258 VJ=100.00  +MOVJ EC00258 VJ=100.00
'Path W939
SFTOF3D
SFTON3D P039
MOVJ C00259 BC00259 VJ=100.00  +MOVJ EC00259 VJ=100.00
SMOVL C00260 BC00260 V=400.0  +MOVJ EC00260
SMOVL C00261 BC00261 V=166.7 PL=0  +MOVJ EC00261
SREFP 1 C00262 BC00262  +REFP EC00262
SREFP 2 C00263 BC00263  +REFP EC00263
MACRO1 MJ#(0) ARGF14
ARCON
SMOVL C00264 BC00264 V=10.0  +MOVJ EC00264
ARCOF
SMOVL C00265 BC00265 V=400.0  +MOVJ EC00265
SMOVL C00266 BC00266 V=1000.0  +MOVJ EC00266
SFTOF3D
MOVJ C00267 BC00267 VJ=100.00  +MOVJ EC00267 VJ=100.00
'Path W941
SFTOF3D
SFTON3D P039
MOVJ C00268 BC00268 VJ=100.00  +MOVJ EC00268 VJ=100.00
SMOVL C00269 BC00269 V=400.0  +MOVJ EC00269
SMOVL C00270 BC00270 V=133.3 PL=0  +MOVJ EC00270
SREFP 1 C00271 BC00271  +REFP EC00271
SREFP 2 C00272 BC00272  +REFP EC00272
ARCON
SMOVL C00273 BC00273 V=10.0  +MOVJ EC00273
ARCOF
SMOVL C00274 BC00274 V=400.0  +MOVJ EC00274
SFTOF3D
SMOVL C00275 BC00275 V=1000.0  +MOVJ EC00275
MOVJ C00276 BC00276 VJ=100.00  +MOVJ EC00276 VJ=10.00
SFTOF3D
MOVJ C00277 BC00277 VJ=100.00  +MOVJ EC00277 VJ=100.00
MOVJ C00278 BC00278 VJ=100.00  +MOVJ EC00278 VJ=15.00
'9
'Path W942
SFTOF3D
SFTON3D P038
MOVJ C00279 BC00279 VJ=100.00  +MOVJ EC00279 VJ=100.00
SMOVL C00280 BC00280 V=166.7 PL=0  +MOVJ EC00280
SREFP 1 C00281 BC00281  +REFP EC00281
SREFP 2 C00282 BC00282  +REFP EC00282
MACRO1 MJ#(0) ARGF14
ARCON
SMOVL C00283 BC00283 V=10.0  +MOVJ EC00283
ARCOF
SFTOF3D
SMOVL C00284 BC00284 V=400.0  +MOVJ EC00284
SMOVL C00285 BC00285 V=1000.0  +MOVJ EC00285
SFTOF3D
'Path W943
SFTOF3D
SFTON3D P038
SMOVL C00286 BC00286 V=133.3 PL=0  +MOVJ EC00286
SREFP 1 C00287 BC00287  +REFP EC00287
SREFP 2 C00288 BC00288  +REFP EC00288
MACRO1 MJ#(0) ARGF14
ARCON
SMOVL C00289 BC00289 V=10.0  +MOVJ EC00289
ARCOF
SMOVL C00290 BC00290 V=400.0  +MOVJ EC00290
SFTOF3D
'Path W944
SFTOF3D
SFTON3D P038
SMOVL C00291 BC00291 V=166.7 PL=0  +MOVJ EC00291
SREFP 1 C00292 BC00292  +REFP EC00292
SREFP 2 C00293 BC00293  +REFP EC00293
MACRO1 MJ#(0) ARGF14
ARCON
SMOVL C00294 BC00294 V=10.0  +MOVJ EC00294
SMOVL C00295 BC00295 V=10.0  +MOVJ EC00295
ARCOF
SMOVL C00296 BC00296 V=400.0  +MOVJ EC00296
SFTOF3D
'10
'11
MOVJ C00297 BC00297 VJ=100.00  +MOVJ EC00297 VJ=100.00
'Path W946
SFTOF3D
SFTON3D P033
SMOVL C00298 BC00298 V=166.7 PL=0  +MOVJ EC00298
SREFP 1 C00299 BC00299  +REFP EC00299
SREFP 2 C00300 BC00300  +REFP EC00300
MACRO1 MJ#(0) ARGF14
ARCON
SMOVL C00301 BC00301 V=10.0  +MOVJ EC00301
SMOVL C00302 BC00302 V=10.0  +MOVJ EC00302
SMOVL C00303 BC00303 V=10.0  +MOVJ EC00303
SMOVL C00304 BC00304 V=10.0  +MOVJ EC00304
ARCOF
SMOVL C00305 BC00305 V=400.0  +MOVJ EC00305
SMOVL C00306 BC00306 V=400.0  +MOVJ EC00306
SMOVL C00307 BC00307 V=1000.0  +MOVJ EC00307
SFTOF3D
'Path W948
SFTOF3D
SFTON3D P033
SMOVL C00308 BC00308 V=166.7 PL=0  +MOVJ EC00308
SREFP 1 C00309 BC00309  +REFP EC00309
SREFP 2 C00310 BC00310  +REFP EC00310
ARCON
SMOVL C00311 BC00311 V=10.0  +MOVJ EC00311
ARCOF
SMOVL C00312 BC00312 V=400.0  +MOVJ EC00312
SMOVL C00313 BC00313 V=400.0  +MOVJ EC00313
SMOVL C00314 BC00314 V=1000.0  +MOVJ EC00314
SFTOF3D
'12
'Path W945
SFTOF3D
SFTON3D P034
MOVJ C00315 BC00315 VJ=100.00  +MOVJ EC00315 VJ=100.00
SMOVL C00316 BC00316 V=400.0  +MOVJ EC00316
SMOVL C00317 BC00317 V=166.7 PL=0  +MOVJ EC00317
SREFP 1 C00318 BC00318  +REFP EC00318
SREFP 2 C00319 BC00319  +REFP EC00319
MACRO1 MJ#(0) ARGF14
ARCON
SWVON WEV#(21)
SMOVL C00320 BC00320 V=9.2  +MOVJ EC00320
ARCOF
SWVOF
SMOVL C00321 BC00321 V=400.0  +MOVJ EC00321
SMOVL C00322 BC00322 V=1000.0  +MOVJ EC00322
SFTOF3D
'Path W949
SFTOF3D
SFTON3D P036
MOVJ C00323 BC00323 VJ=100.00  +MOVJ EC00323 VJ=100.00
SMOVL C00324 BC00324 V=166.7 PL=0  +MOVJ EC00324
SREFP 1 C00325 BC00325  +REFP EC00325
SREFP 2 C00326 BC00326  +REFP EC00326
MACRO1 MJ#(0) ARGF14
ARCON
SMOVL C00327 BC00327 V=10.0  +MOVJ EC00327
SMOVL C00328 BC00328 V=10.0  +MOVJ EC00328
SMOVL C00329 BC00329 V=10.0  +MOVJ EC00329
SMOVL C00330 BC00330 V=10.0  +MOVJ EC00330
ARCOF
SMOVL C00331 BC00331 V=400.0  +MOVJ EC00331
SMOVL C00332 BC00332 V=1000.0  +MOVJ EC00332
SFTOF3D
'Path W950
SFTOF3D
SFTON3D P036
MOVJ C00333 BC00333 VJ=100.00  +MOVJ EC00333 VJ=100.00
SMOVL C00334 BC00334 V=1000.0  +MOVJ EC00334
SFTOF3D
MOVJ C00335 BC00335 VJ=100.00  +MOVJ EC00335 VJ=10.00
MOVJ C00336 BC00336 VJ=100.00  +MOVJ EC00336 VJ=100.00
'Path W951
SFTOF3D
SFTON3D P036
MOVJ C00337 BC00337 VJ=100.00  +MOVJ EC00337 VJ=100.00
SMOVL C00338 BC00338 V=400.0  +MOVJ EC00338
SMOVL C00339 BC00339 V=166.7 PL=0  +MOVJ EC00339
SREFP 1 C00340 BC00340  +REFP EC00340
SREFP 2 C00341 BC00341  +REFP EC00341
MACRO1 MJ#(0) ARGF9
ARCON
SMOVL C00342 BC00342 V=10.0  +MOVJ EC00342
ARCOF
SMOVL C00343 BC00343 V=400.0  +MOVJ EC00343
SMOVL C00344 BC00344 V=1000.0  +MOVJ EC00344
SFTOF3D
MOVJ C00345 BC00345 VJ=100.00  +MOVJ EC00345 VJ=100.00
MOVJ C00346 BC00346 VJ=100.00  +MOVJ EC00346 VJ=100.00
'13
'Path W952
SFTOF3D
SFTON3D P041
SMOVL C00347 BC00347 V=400.0  +MOVJ EC00347
SMOVL C00348 BC00348 V=166.7  +MOVJ EC00348
ARCON
SMOVL C00349 BC00349 V=10.0  +MOVJ EC00349
SMOVL C00350 BC00350 V=10.0  +MOVJ EC00350
ARCOF
SMOVL C00351 BC00351 V=200.0  +MOVJ EC00351
SMOVL C00352 BC00352 V=166.7 PL=0  +MOVJ EC00352
SREFP 1 C00353 BC00353  +REFP EC00353
SREFP 2 C00354 BC00354  +REFP EC00354
MACRO1 MJ#(0) ARGF14
ARCON
SMOVL C00355 BC00355 V=10.8  +MOVJ EC00355
SFTON3D P042
SMOVL C00356 BC00356 V=10.8  +MOVJ EC00356
ARCOF
SMOVL C00357 BC00357 V=400.0  +MOVJ EC00357
SFTOF3D
MOVJ C00358 BC00358 VJ=100.00  +MOVJ EC00358 VJ=10.00
MOVJ C00359 BC00359 VJ=100.00  +MOVJ EC00359 VJ=100.00
SMOVL C00360 BC00360 V=1000.0  +MOVJ EC00360
SFTON3D P055
MACRO1 MJ#(0) ARGF9
SMOVL C00361 BC00361 V=333.3  +MOVJ EC00361
ARCON
SMOVL C00362 BC00362 V=11.7  +MOVJ EC00362
ARCOF
SFTOF3D
SMOVL C00363 BC00363 V=333.3  +MOVJ EC00363
MOVJ C00364 BC00364 VJ=100.00  +MOVJ EC00364 VJ=20.00
MOVJ C00365 BC00365 VJ=100.00  +MOVJ EC00365 VJ=20.00
SFTON3D P060
SMOVL C00366 BC00366 V=166.7  +MOVJ EC00366
ARCON
SMOVL C00367 BC00367 V=11.7  +MOVJ EC00367
ARCOF
SMOVL C00368 BC00368 V=333.3  +MOVJ EC00368
SFTOF3D
MOVJ C00369 BC00369 VJ=100.00  +MOVJ EC00369 VJ=10.00
MOVJ C00370 BC00370 VJ=100.00  +MOVJ EC00370 VJ=10.00
'Path W954
SFTOF3D
SFTON3D P037
MOVJ C00371 BC00371 VJ=100.00  +MOVJ EC00371 VJ=100.00
SMOVL C00372 BC00372 V=400.0  +MOVJ EC00372
SMOVL C00373 BC00373 V=166.7 PL=0  +MOVJ EC00373
SREFP 1 C00374 BC00374  +REFP EC00374
SREFP 2 C00375 BC00375  +REFP EC00375
MACRO1 MJ#(0) ARGF14
ARCON
SMOVL C00376 BC00376 V=10.0  +MOVJ EC00376
SMOVL C00377 BC00377 V=10.0  +MOVJ EC00377
ARCOF
SMOVL C00378 BC00378 V=400.0  +MOVJ EC00378
SMOVL C00379 BC00379 V=1000.0  +MOVJ EC00379
SFTOF3D
'Path W955
SFTOF3D
SFTON3D P037
SMOVL C00380 BC00380 V=400.0  +MOVJ EC00380
SMOVL C00381 BC00381 V=133.3 PL=0  +MOVJ EC00381
SREFP 1 C00382 BC00382  +REFP EC00382
SREFP 2 C00383 BC00383  +REFP EC00383
MACRO1 MJ#(0) ARGF14
ARCON
SMOVL C00384 BC00384 V=10.0  +MOVJ EC00384
ARCOF
SMOVL C00385 BC00385 V=400.0  +MOVJ EC00385
SFTOF3D
MOVJ C00386 BC00386 VJ=100.00  +MOVJ EC00386 VJ=100.00
MOVJ C00387 BC00387 VJ=100.00  +MOVJ EC00387 VJ=50.00
'Path W956
SFTOF3D
SFTON3D P037
MOVJ C00388 BC00388 VJ=100.00  +MOVJ EC00388 VJ=100.00
SMOVL C00389 BC00389 V=400.0  +MOVJ EC00389
SMOVL C00390 BC00390 V=133.3 PL=0  +MOVJ EC00390
SREFP 1 C00391 BC00391  +REFP EC00391
SREFP 2 C00392 BC00392  +REFP EC00392
MACRO1 MJ#(0) ARGF14
ARCON
SMOVL C00393 BC00393 V=10.0  +MOVJ EC00393
ARCOF
SMOVL C00394 BC00394 V=400.0  +MOVJ EC00394
SMOVL C00395 BC00395 V=1000.0  +MOVJ EC00395
SFTOF3D
'17
MOVJ C00396 BC00396 VJ=100.00  +MOVJ EC00396 VJ=100.00
MOVJ C00397 BC00397 VJ=100.00  +MOVJ EC00397 VJ=100.00
'Path W957
SFTOF3D
SFTON3D P040
SMOVL C00398 BC00398 V=166.7 PL=0  +MOVJ EC00398
SREFP 1 C00399 BC00399  +REFP EC00399
SREFP 2 C00400 BC00400  +REFP EC00400
MACRO1 MJ#(0) ARGF14
ARCON
SMOVL C00401 BC00401 V=10.0  +MOVJ EC00401
ARCOF
SMOVL C00402 BC00402 V=400.0  +MOVJ EC00402
SMOVL C00403 BC00403 V=333.3  +MOVJ EC00403
SFTOF3D
'Path W958
SFTOF3D
SFTON3D P040
SMOVL C00404 BC00404 V=166.7 PL=0  +MOVJ EC00404
SREFP 1 C00405 BC00405  +REFP EC00405
SREFP 2 C00406 BC00406  +REFP EC00406
MACRO1 MJ#(0) ARGF14
ARCON
SMOVL C00407 BC00407 V=10.0  +MOVJ EC00407
ARCOF
SMOVL C00408 BC00408 V=400.0  +MOVJ EC00408
SFTOF3D
MOVJ C00409 BC00409 VJ=100.00  +MOVJ EC00409 VJ=100.00
'Path W959
SFTOF3D
SFTON3D P040
COMM MOVJ C00410 BC00410 VJ=100.00  +MOVJ EC00410 VJ=100.00
COMM SMOVL C00411 BC00411 V=400.0  +MOVJ EC00411
COMM SMOVL C00412 BC00412 V=100.0 PL=0  +MOVJ EC00412
COMM SREFP 1 C00413 BC00413  +REFP EC00413
COMM SREFP 2 C00414 BC00414  +REFP EC00414
COMM MACRO1 MJ#(0) ARGF0
COMM ARCON
COMM SMOVL C00415 BC00415 V=10.0  +MOVJ EC00415
COMM SMOVL C00416 BC00416 V=10.0  +MOVJ EC00416
COMM SMOVL C00417 BC00417 V=10.0  +MOVJ EC00417
COMM ARCOF
COMM SMOVL C00418 BC00418 V=400.0  +MOVJ EC00418
COMM SMOVL C00419 BC00419 V=1000.0  +MOVJ EC00419
SFTOF3D
'18
'Path W960
SFTOF3D
MOVJ C00420 BC00420 VJ=100.00  +MOVJ EC00420 VJ=100.00
MOVJ C00421 BC00421 VJ=100.00  +MOVJ EC00421 VJ=15.00
MOVJ C00422 BC00422 VJ=100.00  +MOVJ EC00422 VJ=15.00
SMOVL C00423 BC00423 V=400.0  +MOVJ EC00423
SFTON3D P050
SMOVL C00424 BC00424 V=166.7 PL=0  +MOVJ EC00424
SREFP 1 C00425 BC00425  +REFP EC00425
SREFP 2 C00426 BC00426  +REFP EC00426
MACRO1 MJ#(0) ARGF14
ARCON
SMOVL C00427 BC00427 V=9.2  +MOVJ EC00427
SMOVL C00428 BC00428 V=9.2  +MOVJ EC00428
SMOVL C00429 BC00429 V=9.2  +MOVJ EC00429
SMOVL C00430 BC00430 V=9.2  +MOVJ EC00430
SMOVL C00431 BC00431 V=9.2  +MOVJ EC00431
ARCOF
SMOVL C00432 BC00432 V=400.0  +MOVJ EC00432
SMOVL C00433 BC00433 V=1000.0  +MOVJ EC00433
SFTOF3D
'19
MOVJ C00434 BC00434 VJ=100.00  +MOVJ EC00434 VJ=10.00
MOVJ C00435 BC00435 VJ=100.00  +MOVJ EC00435 VJ=100.00
'Path W962
SFTOF3D
SFTON3D P035
MOVJ C00436 BC00436 VJ=100.00  +MOVJ EC00436 VJ=100.00
SMOVL C00437 BC00437 V=400.0  +MOVJ EC00437
SMOVL C00438 BC00438 V=166.7 PL=0  +MOVJ EC00438
SREFP 1 C00439 BC00439  +REFP EC00439
SREFP 2 C00440 BC00440  +REFP EC00440
ARCON
SWVON WEV#(21)
SMOVL C00441 BC00441 V=9.2  +MOVJ EC00441
ARCOF
SWVOF
SMOVL C00442 BC00442 V=400.0  +MOVJ EC00442
SMOVL C00443 BC00443 V=1000.0  +MOVJ EC00443
SFTOF3D
'20
MOVJ C00444 BC00444 VJ=100.00  +MOVJ EC00444 VJ=100.00
MOVJ C00445 BC00445 VJ=100.00  +MOVJ EC00445 VJ=10.00
MOVJ C00446 BC00446 VJ=100.00  +MOVJ EC00446 VJ=100.00
'Path W963
SFTOF3D
SFTON3D P052
SMOVL C00447 BC00447 V=400.0  +MOVJ EC00447
SMOVL C00448 BC00448 V=166.7 PL=0  +MOVJ EC00448
SREFP 1 C00449 BC00449  +REFP EC00449
SREFP 2 C00450 BC00450  +REFP EC00450
MACRO1 MJ#(0) ARGF6
ARCON
SMOVL C00451 BC00451 V=7.5  +MOVJ EC00451
SMOVL C00452 BC00452 V=7.5  +MOVJ EC00452
SMOVL C00453 BC00453 V=7.5  +MOVJ EC00453
ARCOF
SMOVL C00454 BC00454 V=400.0  +MOVJ EC00454
SFTOF3D
'Path W964
SFTOF3D
SFTON3D P052
SMOVL C00455 BC00455 V=500.0  +MOVJ EC00455
SFTOF3D
SFTON3D P052
SMOVL C00456 BC00456 V=500.0  +MOVJ EC00456
SMOVL C00457 BC00457 V=166.7 PL=0  +MOVJ EC00457
SREFP 1 C00458 BC00458  +REFP EC00458
SREFP 2 C00459 BC00459  +REFP EC00459
MACRO1 MJ#(0) ARGF6
ARCON
SMOVL C00460 BC00460 V=9.2  +MOVJ EC00460
ARCOF
SMOVL C00461 BC00461 V=400.0  +MOVJ EC00461
SMOVL C00462 BC00462 V=1000.0  +MOVJ EC00462
SFTOF3D
'Path W967
SFTOF3D
SFTON3D P052
MOVJ C00463 BC00463 VJ=100.00  +MOVJ EC00463 VJ=10.00
MOVJ C00464 BC00464 VJ=100.00  +MOVJ EC00464 VJ=100.00
SMOVL C00465 BC00465 V=500.0  +MOVJ EC00465
SMOVL C00466 BC00466 V=166.7 PL=0  +MOVJ EC00466
SREFP 1 C00467 BC00467  +REFP EC00467
SREFP 2 C00468 BC00468  +REFP EC00468
MACRO1 MJ#(0) ARGF6
ARCON
SMOVL C00469 BC00469 V=10.0  +MOVJ EC00469
ARCOF
SMOVL C00470 BC00470 V=500.0  +MOVJ EC00470
SFTOF3D
MOVJ C00471 BC00471 VJ=100.00  +MOVJ EC00471 VJ=100.00
'21
MOVJ C00472 BC00472 VJ=100.00  +MOVJ EC00472 VJ=100.00
MOVJ C00473 BC00473 VJ=100.00  +MOVJ EC00473 VJ=100.00
'Path W968
SFTOF3D
SFTON3D P031
SMOVL C00474 BC00474 V=500.0  +MOVJ EC00474
SMOVL C00475 BC00475 V=166.7 PL=0  +MOVJ EC00475
SREFP 1 C00476 BC00476  +REFP EC00476
SREFP 2 C00477 BC00477  +REFP EC00477
MACRO1 MJ#(0) ARGF9
ARCON
SFTON3D P032
SMOVL C00478 BC00478 V=10.8  +MOVJ EC00478
ARCOF
SMOVL C00479 BC00479 V=400.0  +MOVJ EC00479
SFTOF3D
MOVJ C00480 BC00480 VJ=100.00  +MOVJ EC00480 VJ=100.00
MOVJ C00481 BC00481 VJ=100.00  +MOVJ EC00481 VJ=100.00
MOVJ C00482 BC00482 VJ=100.00  +MOVJ EC00482 VJ=100.00
CALL JOB:CLEAN-R1_KM_NEW
'cut_wire_dol
'cut_wire_dol
'cut_wire_dol
MOVJ C00483 BC00483 VJ=100.00  +MOVJ EC00483 VJ=100.00
'Path S1328
SFTOF3D
MOVJ C00484 BC00484 VJ=100.00  +MOVJ EC00484 VJ=100.00
MOVJ C00485 BC00485 VJ=100.00  +MOVJ EC00485 VJ=100.00
MOVJ C00486 BC00486 VJ=15.00  +MOVJ EC00486 VJ=100.00
MOVL C00487 BC00487 V=333.3  +MOVJ EC00487 VJ=100.00
SFTOF3D
SMOVL C00488 BC00488 V=166.7  +MOVJ EC00488
SREFP 3 C00489 BC00489  +REFP EC00489
CALL JOB:SEARCH-R1-S13D
SET P023 P006
SFTON3D P023
SMOVL C00490 BC00490 V=166.7  +MOVJ EC00490
SMOVL C00491 BC00491 V=166.7  +MOVJ EC00491
SMOVL C00492 BC00492 V=166.7  +MOVJ EC00492
SREFP 3 C00493 BC00493  +REFP EC00493
CALL JOB:SEARCH-R1-S13D
SET P023 P006
SFTON3D P023
SMOVL C00494 BC00494 V=166.7  +MOVJ EC00494
MOVL C00495 BC00495 V=400.0  +MOVJ EC00495 VJ=100.00
MOVJ C00496 BC00496 VJ=100.00  +MOVJ EC00496 VJ=100.00
MOVJ C00497 BC00497 VJ=100.00  +MOVJ EC00497 VJ=100.00
'Path S1331
SFTOF3D
MOVL C00498 BC00498 V=166.7  +MOVJ EC00498 VJ=100.00
SMOVL C00499 BC00499 V=166.7  +MOVJ EC00499
SREFP 3 C00500 BC00500  +REFP EC00500
CALL JOB:SEARCH-R1-S13D
SET P022 P006
SFTON3D P022
SMOVL C00501 BC00501 V=166.7  +MOVJ EC00501
SMOVL C00502 BC00502 V=166.7  +MOVJ EC00502
SMOVL C00503 BC00503 V=166.7  +MOVJ EC00503
SREFP 3 C00504 BC00504  +REFP EC00504
CALL JOB:SEARCH-R1-S13D
SET P022 P006
SFTON3D P022
SFTOF3D
SMOVL C00505 BC00505 V=166.7  +MOVJ EC00505
MOVL C00506 BC00506 V=400.0  +MOVJ EC00506 VJ=100.00
MOVJ C00507 BC00507 VJ=100.00  +MOVJ EC00507 VJ=100.00
MOVJ C00508 BC00508 VJ=100.00  +MOVJ EC00508 VJ=100.00
MOVJ C00509 BC00509 VJ=50.00  +MOVJ EC00509 VJ=100.00
MOVJ C00510 BC00510 VJ=100.00  +MOVJ EC00510 VJ=100.00
MOVJ C00511 BC00511 VJ=100.00  +MOVJ EC00511 VJ=100.00
MOVJ C00512 BC00512 VJ=10.00  +MOVJ EC00512 VJ=100.00
MOVJ C00513 BC00513 VJ=100.00  +MOVJ EC00513 VJ=100.00
SMOVL C00514 BC00514 V=166.7  +MOVJ EC00514
SREFP 3 C00515 BC00515  +REFP EC00515
CALL JOB:SEARCH-R1-S13D
SET P030 P006
SFTON3D P030
SMOVL C00516 BC00516 V=166.7  +MOVJ EC00516
SMOVL C00517 BC00517 V=166.7  +MOVJ EC00517
SMOVL C00518 BC00518 V=166.7  +MOVJ EC00518
SREFP 3 C00519 BC00519  +REFP EC00519
CALL JOB:SEARCH-R1-S13D
SET P030 P006
SFTON3D P030
SMOVL C00520 BC00520 V=166.7  +MOVJ EC00520
SFTOF3D
SMOVL C00521 BC00521 V=166.7  +MOVJ EC00521
SMOVL C00522 BC00522 V=166.7  +MOVJ EC00522
SMOVL C00523 BC00523 V=166.7  +MOVJ EC00523
SREFP 3 C00524 BC00524  +REFP EC00524
CALL JOB:SEARCH-R1-S13D
SET P031 P006
SFTON3D P031
SMOVL C00525 BC00525 V=166.7  +MOVJ EC00525
SREFP 3 C00526 BC00526  +REFP EC00526
CALL JOB:SEARCH-R1-S13D
SET P031 P006
SFTON3D P031
SMOVL C00527 BC00527 V=166.7  +MOVJ EC00527
MOVL C00528 BC00528 V=333.3  +MOVJ EC00528 VJ=100.00
'Path S1333
SFTOF3D
MOVJ C00529 BC00529 VJ=40.00  +MOVJ EC00529 VJ=100.00
MOVJ C00530 BC00530 VJ=100.00  +MOVJ EC00530 VJ=100.00
MOVJ C00531 BC00531 VJ=100.00  +MOVJ EC00531 VJ=100.00
MOVJ C00532 BC00532 VJ=100.00  +MOVJ EC00532 VJ=100.00
MOVJ C00533 BC00533 VJ=100.00  +MOVJ EC00533 VJ=100.00
MOVJ C00534 BC00534 VJ=100.00  +MOVJ EC00534 VJ=100.00
MOVJ C00535 BC00535 VJ=100.00  +MOVJ EC00535 VJ=100.00
MOVJ C00536 BC00536 VJ=100.00  +MOVJ EC00536 VJ=100.00
MOVJ C00537 BC00537 VJ=100.00  +MOVJ EC00537 VJ=100.00
MOVL C00538 BC00538 V=400.0  +MOVJ EC00538 VJ=100.00
SMOVL C00539 BC00539 V=166.7  +MOVJ EC00539
SREFP 3 C00540 BC00540  +REFP EC00540
CALL JOB:SEARCH-R1-S13D
SET P021 P006
SFTON3D P021
SMOVL C00541 BC00541 V=166.7  +MOVJ EC00541
SREFP 3 C00542 BC00542  +REFP EC00542
CALL JOB:SEARCH-R1-S13D
SET P021 P006
SFTON3D P021
SMOVL C00543 BC00543 V=166.7  +MOVJ EC00543
'1
'Path W1334
SFTOF3D
SFTON3D P021
SMOVL C00544 BC00544 V=166.7 PL=0  +MOVJ EC00544
SREFP 1 C00545 BC00545  +REFP EC00545
SREFP 2 C00546 BC00546  +REFP EC00546
MACRO1 MJ#(0) ARGF9
SMOVL C00547 BC00547 V=166.7 PL=0  +MOVJ EC00547
ARCON
SMOVL C00548 BC00548 V=12.5  +MOVJ EC00548
ARCOF
SMOVL C00549 BC00549 V=400.0  +MOVJ EC00549
SFTOF3D
MOVJ C00550 BC00550 VJ=100.00  +MOVJ EC00550 VJ=100.00
MOVJ C00551 BC00551 VJ=100.00  +MOVJ EC00551 VJ=100.00
MOVJ C00552 BC00552 VJ=100.00  +MOVJ EC00552 VJ=10.00
'2
'Path W1338
SFTOF3D
MOVJ C00553 BC00553 VJ=100.00  +MOVJ EC00553 VJ=10.00
MOVJ C00554 BC00554 VJ=50.00  +MOVJ EC00554 VJ=10.00
SFTON3D P023
